// TwinCAT 3 PLC project Steinemann
// Title: CalmarProductSteinemann
// Company: WIFAG-Polytype
// Author: Wifag//Polytype
// ProjectVersion: 3.0.4
// Description: All rights reserved (c) Wifag//Polytype, Fribourg/Switzerland (2021)
// ProgramVersion: 3.1.4023.0
// CompilerDefines: checks_in_libs
// libraries:
//   CalmarCommons, * (WIFAG-Polytype)
//   CalmarCompDevices, * (WIFAG-Polytype)
//   CalmarCompInkSystem, * (WIFAG-Polytype)
//   CalmarCompPrint, * (WIFAG-Polytype)
//   CalmarCompSystem, * (WIFAG-Polytype)
//   CalmarCompTcpIp, * (WIFAG-Polytype)
//   CmpBitmapPool, * (System)
//   Tc2_EtherCAT, * (Beckhoff Automation GmbH)
//   Tc2_Math, * (Beckhoff Automation GmbH)
//   Tc2_Standard, * (Beckhoff Automation GmbH)
//   Tc2_System, * (Beckhoff Automation GmbH)
//   Tc2_TcpIp, * (Beckhoff Automation GmbH)
//   Tc2_Utilities, * (Beckhoff Automation GmbH)
//   Tc3_JsonXml, * (Beckhoff Automation GmbH)
//   VisuDialogs, * (System)
// project tree:
//   DUTs/ADS/ ST_ADS_CLEAN_AXIS.TcDUT, ST_ADS_CLEAN_PROCESS.TcDUT, ST_ADS_DFOIL.TcDUT, ST_ADS_DRYER.TcDUT, ST_ADS_DVTSHEETALIGNMENT.TcDUT, ST_ADS_MOTION_CONTROLLER.TcDUT, ST_ADS_MOTION_SYSTEM.TcDUT, ST_ADS_MOTION_XYR_CONTROLLER.TcDUT, ST_ADS_MOTION_XYR_SYSTEM.TcDUT, ST_ADS_SECURITY.TcDUT
//   DUTs/Camera/ EN_CAMERA_TEACH.TcDUT, E_CameraDevice.TcDUT, E_CameraMode.TcDUT, E_DeformationType.TcDUT, ST_ADS_CAMERA.TcDUT, ST_CameraPoint.TcDUT, ST_CAMERA_CORRECTION_QV.TcDUT, ST_CAMERA_RESULT.TcDUT, ST_CAMERA_TEACH_QV.TcDUT, ST_CORRECTION_POINT.TcDUT, ST_TeachPoint.TcDUT
//   DUTs/CleaningStation/ EN_CLEANING_OP.TcDUT, EN_Cleaning_State.TcDUT, EN_EL7201_STATE.TcDUT, EN_EL7342_STATE.TcDUT, ST_CH_MVT_STATUS.TcDUT, ST_CLEANING_DEV_CMD.TcDUT, ST_CLEANING_DEV_STATUS.TcDUT, ST_CU_STATUS.TcDUT, ST_MANUAL_CMD.TcDUT, ST_PU_STATUS.TcDUT, ST_SPEEDS.TcDUT
//   DUTs/ EN_MSG_LIST.TcDUT, ST_DFOIL_RECORD.TcDUT, ST_SENSOR_COMPARISON.TcDUT
//   / GlobalTextList.TcGTLO, ImagePool_Steinemann.TcIPO (not stored), Visualization Manager.TcVMO (not stored)
//   GVLs/ EC_DefGrid.TcGVL, GVL_Camera.TcGVL, GVL_Deformation.TcGVL, GVL_WEU.TcGVL, GVL_Maxliner.TcGVL
//   POUs/Machine/CleaningStation/ADS/ FB_ADS_CleanAxis.TcPOU, FB_ADS_CleanProcess.TcPOU
//   POUs/Machine/CleaningStation/ FB_CappingCommand.TcPOU, FB_CH_MOTION_CTRL.TcPOU, FB_CH_PROCESS_CTRL.TcPOU, FB_CleanDevice.TcPOU, FB_CleaningMotorAxisCH.TcPOU, FB_CleaningMotorAxisCU.TcPOU, FB_CleaningMotorAxisPU.TcPOU, FB_CleaningProcess.TcPOU, FB_CleaningProcessStateBase.TcPOU, FB_CleaningProcessStateCapping.TcPOU, FB_CleaningProcessStateCappingExit.TcPOU, FB_CleaningProcessStateCleaning.TcPOU, FB_CleaningProcessStateError.TcPOU, FB_CleaningProcessStateInit.TcPOU, FB_CleaningProcessStateProduction.TcPOU, FB_CleaningProcessStateService.TcPOU, FB_CleaningProcessStateWait.TcPOU, FB_CLEANING_PROCESS.TcPOU, FB_Cleaning_ValvePump.TcPOU, FB_CU_MOTION_CTRL.TcPOU, FB_EL7041.TcPOU, FB_EL7201.TcPOU, FB_EL7201_001_AXIS_CTRL.TcPOU, FB_EL7201_AXIS_CTRL.TcPOU, FB_EL7342_AXIS_CTRL.TcPOU, FB_MachineBase.TcPOU, FB_MachineState.TcPOU, FB_MOTOR_SWITCH.TcPOU, FB_PU_MOTION_CTRL.TcPOU, FB_SHUTTER.TcPOU, I_CleanDevice.TcIO, I_CleaningStateCallback.TcIO, I_MachineState.TcIO, I_MachineStateBase.TcIO, _VISU_CleanCH.TcVIS, _VISU_CleanCU.TcVIS, _VISU_CleanProcess.TcVIS, _VISU_CleanPU.TcVIS, _VISU_CleanSequence.TcVIS
//   POUs/Machine/EffectiveEncoderResolutionDetection/ FB_EffectiveEncoderResolutionDetection.TcPOU, _VISU_EffectiveEncoderResolutionDetection.TcVIS
//   POUs/Machine/ExhaustSystem/ FB_ExhaustSystemPrint.TcPOU, _VISU_ExhaustSystemPrint.TcVIS
//   POUs/Machine/ FB_FILTER_MAV_1000.TcPOU, FB_TempLogging_OpcUa.TcPOU
//   POUs/Machine/PowerControl/ FB_PowerControl.TcPOU, _VISU_PowerControl.TcVIS
//   POUs/Machine/SheetDetectSupervision/ FB_SheetDetectSupervision.TcPOU, ST_SheetDetectSupervisionPar.TcDUT (not stored), VISU_SheetDetectSupervision.TcVIS
//   POUs/Machine/UV_LED_Modul/ FB_UvLedModule.TcPOU, _VISU_UvLedModule.TcVIS
//   POUs/Print/Ads/ FB_ADS_CAMERA.TcPOU, FB_ADS_DVTSHEETALIGNMENT.TcPOU
//   POUs/Print/Camera/ FB_CameraBase.TcPOU, FB_CameraDummy.TcPOU, FB_CameraTcpIp.TcPOU, FB_CameraTrigger.TcPOU, FB_MarkCamera.TcPOU, FB_SystronCamera.TcPOU, FB_TcpIpComm.TcPOU, F_DeformationPointAcc_ToString.TcPOU, F_CamPoint_ToString.TcPOU, ImagePool.TcIPO (not stored), I_Camera.TcIO, I_CameraSink.TcIO, I_CameraTrigger.TcIO, I_CameraTriggerDevice.TcIO, _VISU_CameraBase.TcVIS, _VISU_CameraBaseSetting.TcVIS, _VISU_CameraTcpIp.TcVIS, _VISU_CameraTcpIpSetting.TcVIS, _VISU_CameraTrigger.TcVIS, _VISU_DeformationPoint.TcVIS, _VISU_MarkCamera.TcVIS (not stored), _VISU_SystronCamera.TcVIS
//   POUs/Print/Camera/LineCamera/ FB_LineCamera.TcPOU, FB_LineCamera106.TcPOU, FB_LineCamera76.TcPOU, FB_LineCamera585.TcPOU, _VISU_LineCamera.TcVIS
//   POUs/Print/Camera/MarkCameraWEU/ E_MarkMode.TcTLEO, FB_MarkCamera_WEU.TcPOU, FB_MarkDefinition.TcPOU, FB_MarkDetection.TcPOU, I_MarkDefinition.TcIO (not stored), ST_MarkDefinition.TcDUT (not stored), ST_MarkState.TcDUT, ST_MarkView.TcDUT (not stored), ST_RepeatHistory.TcDUT (not stored), TL_MarkMode.TcTLO (not stored), _VISU_MarkCamera_WEU.TcVIS, _VISU_MarkDefinition.TcVIS, _VISU_MarkDefinition_Details.TcVIS (not stored), _VISU_MarkDetection.TcVIS, _VISU_MarkDetection_Trigger.TcVIS (not stored), _VISU_MarkHistory.TcVIS, _VISU_MarkHistoryEntry.TcVIS, _VISU_MarkModes.TcVIS, _VISU_MarkOrientation.TcVIS (not stored), _VISU_MarkOverview.TcVIS, _VISU_MarkTriangle.TcVIS (not stored), _VISU_MarkTriangle_Detail.TcVIS (not stored), _VISU_MarkViewMini.TcVIS, _VISU_RepeatHistory.TcVIS (not stored), _VISU_RepeatHistoryEntry.TcVIS
//   POUs/Print/Camera/Obsolete/ FB_CAMERA_TRIGGER.TcPOU
//   POUs/Print/DefGrid/ E_DeformationStep.TcTLEO, FB_ContainerDefGrid.TcPOU, FB_CTManagerDefGrid.TcPOU, FB_CTTrackerView.TcPOU, FB_DeformationPointFIFO.TcPOU, FB_DropSpeedComp.TcPOU, FB_FineAlignement.TcPOU, FB_ImageDeformation.TcPOU, FB_DefGridParamMediator.TcPOU, FB_PointCorr.TcPOU, FB_PrintOverview.TcPOU, FB_PrintPositionDmax.TcPOU, FB_ProdManager_DMAX.TcPOU, FB_PythonDeformation.TcPOU, FB_PythonInterface.TcPOU, FB_GridDataExporter.TcPOU, FB_StartPositionDummy.TcPOU, FB_WorkerDefGrid.TcPOU, FB_WorkerDefGrid_Camera.TcPOU, FB_WorkerDefGrid_Deformation.TcPOU, FB_WorkerDefGrid_Delete.TcPOU, FB_WorkerDefGrid_Inspection.TcPOU, FB_WorkerDefGrid_Print.TcPOU, FB_WorkerDefGrid_Python.TcPOU, FB_WorkerDefGrid_Verify.TcPOU, F_EncoderSpeedComp.TcPOU, F_MeterToSubPixelReal.TcPOU (not stored), I_DeformationHandler.TcIO, I_GridPointCorrection.TcIO, I_Module.TcIO, I_ParamMediator.TcIO, I_ProdManager.TcIO, ST_CameraGridSettings.TcDUT, ST_CameraPointTbl.TcDUT (not stored), ST_DeformationPointTbl.TcDUT, ST_GridPointUI.TcDUT, ST_WorkerDefGrid_CTData.TcDUT
//   POUs/Print/DefGrid/_Test/ E_GridTypeSelection.TcTLEO, Txt_GridTypeSelection.TcTLO
//   POUs/Print/DefGrid/_VISU_Templates/ E_DeformationType.TcTLO, _VISU_ContainerDefGrid.TcVIS, _VISU_CTsFlow.TcVIS, _VISU_CTTrackerFlow.TcVIS, _VISU_CT_Details.TcVIS, _VISU_DefGridTable.TcVIS, _VISU_DefGridTable_raw.TcVIS, _VISU_FineAlignment.TcVIS, _VISU_GridPointView.TcVIS (not stored), _VISU_ImageDeformation.TcVIS (not stored), _VISU_PlacementXY.TcVIS (not stored), _VISU_PlacementXY_puc.TcVIS (not stored), _VISU_PlacementXY_cross.TcVIS (not stored), _VISU_PmPosition.TcVIS (not stored), _VISU_PrintPositionDmax.TcVIS (not stored), _VISU_DropSpeedComp_Setup.TcVIS, _VISU_ProductionOverview.TcVIS (not stored), _VISU_StartPositionDummy.TcVIS (not stored), _VISU_WorkerDefGrid.TcVIS (not stored), _VISU_WorkerDefGrid_Camera.TcVIS (not stored), _VISU_WorkerDefGrid_Deformation.TcVIS (not stored), _VISU_WorkerDefGrid_Delete.TcVIS (not stored), _VISU_WorkerDefGrid_Print.TcVIS (not stored), _VISU_WorkerDefGrid_Python.TcVIS (not stored), _VISU_WorkerDefGrid_small.TcVIS (not stored), _VISU_WorkerDefGrid_Verify.TcVIS (not stored), _VISU_WorkerDefGrid_VerifyDetail.TcVIS (not stored), _VISU_CTGridExporter.TcVIS, _VISU_WorkerDefGrid_VerifyHistory.TcVIS (not stored)
//   POUs/Print/Global/ I_PrintGlobal.TcIO
//   POUs/Print/Maxliner/ FB_PrintModule_Maxliner.TcPOU, FB_PrintModule_Maxliner_View.TcPOU, _VISU_PmEnable_Maxliner.TcVIS, _VISU_Pm_Maxliner_ImgLengthCheck.TcVIS, _VISU_Pm_Maxliner_Worker.TcVIS, _VISU_Pm_Maxliner_mini_Worker.TcVIS, _VISU_Pm_Maxliner_Debug.TcVIS, _VISU_Pm_Maxliner.TcVIS, _VISU_Pm_Maxliner_Settings.TcVIS
//   POUs/Print/Module/ FB_PrintModule_Base.TcPOU, ST_CassetteSetup.TcDUT, ST_CassetteSetup_Ink.TcDUT, ST_CassetteSetup_Print.TcDUT, ST_MappingDefinition.TcDUT, ST_ModuleMachineInterface_IN.TcDUT, ST_ModuleMachineInterface_OUT.TcDUT
//   POUs/Print/Module/_VISU_Templates/ _VISU_PmEnable.TcVIS (not stored), _VISU_PmEnable_1Worker.TcVIS (not stored), _VISU_Pm_Base_Settings.TcVIS (not stored), _VISU_Pm_MachineIn.TcVIS (not stored), _VISU_Pm_MachineOut.TcVIS (not stored)
//   POUs/Print/obsolete/ FB_DRIFTCONTROL.TcPOU, FB_START_POS_DETECT_WEU.TcPOU, ST_CassetteSetup_PrintAds.TcDUT (excluded from build)
//   POUs/Print/WEU/ FB_PrintModule_WEU.TcPOU, FB_PrintModule_WEU_View.TcPOU, FB_WorkerDefGrid_Print_WEU.TcPOU, _VISU_PmImgLengthCheck.TcVIS, _VISU_Pm_WEU_Debug.TcVIS, _VISU_Pm_WEU_Settings.TcVIS, _VISU_Pm_WEU.TcVIS, _VISU_Pm_WEU_1Worker.TcVIS, _VISU_Pm_WEU_mini.TcVIS, _VISU_Pm_WEU_mini_1Worker.TcVIS, _VISU_Pm_WEU_Worker.TcVIS, _VISU_WorkerPrint_WEU.TcVIS
//   Version/ Global_Version.TcGVL

// ---- DUTs/ADS/ST_ADS_CLEAN_AXIS.TcDUT
TYPE ST_ADS_CLEAN_AXIS :
(*************************************************************************************************)
(*  FILENAME:    ST_ADS_CLEAN_AXIS.EXP                                                           *)
(*  PROJECT:     CALMAR PUPLC                                                                    *)
(*  COPYRIGHT:   All rights reserved (c) Wifag//Polytype, Fribourg/Switzerland (2016)            *)
(*  ENVIRONMENT: TwinCAT PLC                                                                     *)
(*  VERSION:     <version>                                                                       *)
(*************************************************************************************************)
(*  DESCRIPTION:                                                                   <description> *)
(*     User commands from ADS and info feedback to ADS  for cleaning station axis.               *)
(*                                                                                </description> *)
(*************************************************************************************************)

STRUCT
  iO_Version            : INT :=  010001;   (*1.0.1*)
  aO_Type               : STRING := 'Axis';
  aO_Name               : STRING := '';
  sO_Message            : ST_ADS_MSG_IF;

  bI_FaultAck           : BOOL := FALSE;

  (*Manual Move, only possible when in maintenance and manual mode*)
  bI_ManualMove         : BOOL := FALSE;  (*Active as long as true*)
  bO_ManualMoveCanEx    : BOOL := FALSE;
  bO_ManualMovekExec    : BOOL := FALSE;
  fI_ManualTargetPos    : REAL := 0.0;

  (*Current axis position*)
  sO_AxisPosition       : ST_VAR_OUT_REAL;

  wO_ErrorCode          : WORD;
  bO_Busy               : BOOL;
  bO_Ready              : BOOL;
  bO_Error              : BOOL;
END_STRUCT
END_TYPE

// ---- DUTs/ADS/ST_ADS_CLEAN_PROCESS.TcDUT
TYPE ST_ADS_CLEAN_PROCESS :
(*************************************************************************************************)
(*  FILENAME:    ST_ADS_CLEAN_PROCESS                                                            *)
(*  PROJECT:     CALMAR PUPLC                                                                    *)
(*  COPYRIGHT:   All rights reserved (c) Wifag//Polytype, Fribourg/Switzerland (2016)            *)
(*  ENVIRONMENT: TwinCAT PLC                                                                     *)
(*  VERSION:     <version>                                                                       *)
(*************************************************************************************************)
(*  DESCRIPTION:                                                                   <description> *)
(*     User commands from ADS and info feedback to ADS for cleaning station axis.                *)
(*                                                                                </description> *)
(*************************************************************************************************)

STRUCT
  iO_Version                 : INT :=  010001;  (*1.0.1*)
  aO_Type                    : STRING := 'CleanProcess';
  aO_Name                    : STRING :='';
  sO_Message                 : ST_ADS_MSG_IF;
                             
  (*User commands - Trigger operation*)
  bI_StartCapping            : BOOL := FALSE;
  bO_StartCappingCanEx       : BOOL := FALSE;
  bO_StartCappingExec        : BOOL := FALSE;
                             
  bI_StopCapping             : BOOL := FALSE;
  bO_StopCappingCanEx        : BOOL := FALSE;
  bO_StopCappingExec         : BOOL := FALSE;
                             
  bI_Purge                   : BOOL := FALSE;
  bO_PurgeCanEx              : BOOL := FALSE;
  bO_PurgeExec               : BOOL := FALSE;
                             
  bI_Clean                   : BOOL := FALSE;
  bO_CleanCanEx              : BOOL := FALSE;
  bO_CleanExec               : BOOL := FALSE;
                             
  bI_Maintenance             : BOOL := FALSE;
  bO_MaintenanceCanEx        : BOOL := FALSE;
  bO_MaintenanceExec         : BOOL := FALSE;
                             
  bI_OpenShutter             : BOOL := FALSE;
  bO_OpenShutterCanEx        : BOOL := FALSE;
  bO_OpenShutterExec         : BOOL := FALSE;
                             
  bI_Abort                   : BOOL := FALSE;
  bO_AbortCanEx              : BOOL := FALSE;
  bO_AbortExec               : BOOL := FALSE;

  bI_AcknowledgeError        : BOOL := FALSE;
  bO_AcknowledgeErrorCanEx   : BOOL := FALSE;
  bO_AcknowledgeErrorExec    : BOOL := FALSE;

  (*User settings - State operation*)
  bI_AutoMode                : BOOL := TRUE;  (*del*)
  bI_CleanAfterCapp          : BOOL := FALSE;
  bI_CleanAfterPurge         : BOOL := FALSE;
  bI_PurgeAfterCapp          : BOOL := FALSE; (*del*)
  bI_MaintenanceMode         : BOOL := FALSE;
                             
  (*Flags*)                  
  bO_Busy                    : BOOL;
  bO_Ready                   : BOOL;
  bO_ServiceEnabled          : BOOL;
  bO_AxisProcessMovingVisible: BOOL := TRUE;  (*Cleaning process axis moving is shown at PUC*)
                             
  (*Message Queue - TODO update*)
  bI_FaultAck                : BOOL := FALSE;
  wO_ErrorCode               : WORD;
END_STRUCT
END_TYPE

// ---- DUTs/ADS/ST_ADS_DFOIL.TcDUT
TYPE ST_ADS_DFOIL :
(*************************************************************************************************)
(*  FILENAME:    ST_ADS_DFOIL                                                                    *)
(*  PROJECT:     CALMAR PUPLC                                                                    *)
(*  COPYRIGHT:   All rights reserved (c) Wifag//Polytype, Fribourg/Switzerland (2019)            *)
(*  ENVIRONMENT: TwinCAT PLC                                                                     *)
(*  VERSION:     <version>                                                                       *)
(*************************************************************************************************)
(*  DESCRIPTION:                                                                   <description> *)
(*    ADS structure dFoil system.                                                                *)
(*                                                                                </description> *)
(*************************************************************************************************)

STRUCT
  iO_Version         : INT    := 010000;  (*1.0.0*)
  aO_Type            : STRING := 'dFoil';
  aO_Name            : STRING := 'dFoil';

  bI_Enable          : BOOL := TRUE;      (*Enable this device*)
  iO_MaxNbRecords    : UINT  := SIZEOF(sI_dFoilUsagePos) / SIZEOF(sI_dFoilUsagePos[1]);

  iI_UsedNbRecords   : UINT;
  sI_dFoilUsagePos   : ARRAY[1..20] OF ST_DFOIL_RECORD;
END_STRUCT
END_TYPE

// ---- DUTs/ADS/ST_ADS_DRYER.TcDUT
TYPE ST_ADS_DRYER :
(*************************************************************************************************)
(*  FILENAME:    ST_ADS_DRYER.EXP                                                                *)
(*  PROJECT:     CALMAR PUPLC                                                                    *)
(*  COPYRIGHT:   All rights reserved (c) Wifag//Polytype, Fribourg/Switzerland (2016)            *)
(*  ENVIRONMENT: TwinCAT PLC                                                                     *)
(*  VERSION:     <version>                                                                       *)
(*************************************************************************************************)
(*  DESCRIPTION:                                                                   <description> *)
(*     ADS structure for dryer.                                                                  *)
(*                                                                                </description> *)
(*************************************************************************************************)

STRUCT
  iO_Version                  : INT    := 010001;             (*1.0.1*)
  aO_Type                     : STRING := 'Dryer';
  aO_Name                     : STRING := 'DRYER';
  sO_Message                  : ST_ADS_MSG_IF;                (*Messaging*)

  (*I*)
  bI_Enable                   : BOOL := TRUE;                 (*Enable this device*)

  sI_PositionX                : ST_VAR_IN_DINT;               (*Actual position of the dryer on the axis, in micro meters*)
  sI_StartPositionX           : ST_VAR_IN_DINT;               (*Actual position of the dryer on the axis, in micro meters*)

  (*O*)
  cO_StatusDryer              : BYTE;                         (*Bit0:  1h: exist
                                                                Bit1:  2h: enabled
                                                                Bit2:  4h: dryer activ
                                                                Bit3:  8h: warning
                                                                Bit4: 10h: error*)
END_STRUCT
END_TYPE

// ---- DUTs/ADS/ST_ADS_DVTSHEETALIGNMENT.TcDUT
TYPE ST_ADS_DVTSHEETALIGNMENT :
(*************************************************************************************************)
(*  FILENAME:     ST_ADS_DVTSHEETALIGNMENT.EXP                                                   *)
(*  PROJECT:      CALMAR Print System                                                            *)
(*  COPYRIGHT:    Wifag//Polytype Fribourg                                                       *)
(*  ENVIRONMENT:  TwinCAT PLC / CoDeSys                                                          *)
(*  VERSION:      1.0                                                                            *)
(*  DESCRIPTION:  User settings for DVT sheet alignment                                          *)
(*                                                                                               *)
(*  AUTHOR:       FAF                                                                            *)
(*************************************************************************************************)
(*  MODIFICATIONS:                                                                               *)
(*************************************************************************************************)
(*  Date      Author  Comments                                                                   *)
(*  30.04.14  FAF     Created for general use                                                    *)
(*                                                                                               *)
(*************************************************************************************************)

STRUCT
  iO_Version         : INT :=  010010;  (*1.0.10*)
  aO_Type            : STRING := 'DvtSheetAlignment';
  aO_Name            : STRING :='';
  sO_Message         : ST_ADS_MSG_IF;

  (*In*)
  bI_Enable          : BOOL := FALSE;   (*Enable processing*)

  bI_UsePrintMark    : BOOL := TRUE;    (*Enable processing of print marks*)
  sI_PrintMarkSizeX  : ST_VAR_IN_REAL;  (*Print mark X size [mm]*)
  sI_PrintMarkSizeY  : ST_VAR_IN_REAL;  (*Print mark Y size [mm]*)

  sI_HeadGap         : ST_VAR_IN_REAL;  (*Gap between head and substrate [mm]*)

  lI_SegmentSize     : UDINT;           (*Distance between two images in pixel*)
  lI_SegmentCount    : UDINT;           (*Number of images*)
  fI_SegmentAngle    : REAL;            (*Angle between two segments in deg*)

  sI_DeltaX          : ST_VAR_IN_REAL;  (*X offset between camera marks [mm]*)

  bI_IsMaintenanceJob: BOOL;            (*Maintenance job: disable shift and rotation*)

  (*Out*)
  sO_CurrentAngle    : ST_VAR_OUT_REAL; (*Last measured angle in deg*)
  lO_CurrentYShift   : UDINT;           (*Last measured Y Shift in Pixel*)

  bO_RangeErrorAngle : BOOL;            (*Measured angle out of range*)
  bO_RangeErrorShift : BOOL;            (*Measured shift out of range*)
END_STRUCT
END_TYPE

// ---- DUTs/ADS/ST_ADS_MOTION_CONTROLLER.TcDUT
TYPE ST_ADS_MOTION_CONTROLLER :
(*************************************************************************************************)
(*  FILENAME:    ST_ADS_MOTION_CONTROLLER.EXP                                                    *)
(*  PROJECT:     CALMAR PUPLC                                                                    *)
(*  COPYRIGHT:   All rights reserved (c) Wifag//Polytype, Fribourg/Switzerland (2016)            *)
(*  ENVIRONMENT: TwinCAT PLC                                                                     *)
(*  VERSION:     <version>                                                                       *)
(*************************************************************************************************)
(*  DESCRIPTION:                                                                   <description> *)
(*     Add description                                                                           *)
(*                                                                                </description> *)
(*************************************************************************************************)

STRUCT
  iO_Version        : INT :=  010000;  (*1.0.0*)
  aO_Type           : STRING := 'MotionController';
  aO_Name           : STRING := 'MotionController';

END_STRUCT
END_TYPE

// ---- DUTs/ADS/ST_ADS_MOTION_SYSTEM.TcDUT
TYPE ST_ADS_MOTION_SYSTEM :
(*************************************************************************************************)
(*  FILENAME:    ST_ADS_MOTION_SYSTEM.EXP                                                        *)
(*  PROJECT:     CALMAR PUPLC                                                                    *)
(*  COPYRIGHT:   All rights reserved (c) Wifag//Polytype, Fribourg/Switzerland (2016)            *)
(*  ENVIRONMENT: TwinCAT PLC                                                                     *)
(*  VERSION:     <version>                                                                       *)
(*************************************************************************************************)
(*  DESCRIPTION:                                                                   <description> *)
(*     Add description                                                                           *)
(*                                                                                </description> *)
(*************************************************************************************************)

STRUCT
  iO_Version        : INT :=  010000;  (*1.0.0*)
  aO_Type           : STRING := 'MotionSystem';
  aO_Name           : STRING := 'MotionSystem';

END_STRUCT
END_TYPE

// ---- DUTs/ADS/ST_ADS_MOTION_XYR_CONTROLLER.TcDUT
TYPE ST_ADS_MOTION_XYR_CONTROLLER :
(*************************************************************************************************)
(*  FILENAME:    ST_ADS_MOTION_XYR_CONTROLLER.EXP                                                *)
(*  PROJECT:     CALMAR PUPLC                                                                    *)
(*  COPYRIGHT:   All rights reserved (c) Wifag//Polytype, Fribourg/Switzerland (2016)            *)
(*  ENVIRONMENT: TwinCAT PLC                                                                     *)
(*  VERSION:     <version>                                                                       *)
(*************************************************************************************************)
(*  DESCRIPTION:                                                                   <description> *)
(*     Add description                                                                           *)
(*                                                                                </description> *)
(*************************************************************************************************)

STRUCT
  iO_Version        : INT :=  010000;  (*1.0.0*)
  aO_Type           : STRING := 'MotionXyrController';
  aO_Name           : STRING := 'MotionXYRController';

  aO_IpAddress      : STRING;

END_STRUCT
END_TYPE

// ---- DUTs/ADS/ST_ADS_MOTION_XYR_SYSTEM.TcDUT
TYPE ST_ADS_MOTION_XYR_SYSTEM :
(*************************************************************************************************)
(*  FILENAME:    ST_ADS_MOTION_XYR_SYSTEM.EXP                                                    *)
(*  PROJECT:     CALMAR PUPLC                                                                    *)
(*  COPYRIGHT:   All rights reserved (c) Wifag//Polytype, Fribourg/Switzerland (2016)            *)
(*  ENVIRONMENT: TwinCAT PLC                                                                     *)
(*  VERSION:     <version>                                                                       *)
(*************************************************************************************************)
(*  DESCRIPTION:                                                                   <description> *)
(*     Add description                                                                           *)
(*                                                                                </description> *)
(*************************************************************************************************)

STRUCT
  iO_Version        : INT :=  010000;  (*1.0.0*)
  aO_Type           : STRING := 'MotionXyrSystem';
  aO_Name           : STRING := 'MotionXYRSystem';

  iO_Elevation      : DINT;
  iO_Rotation       : DINT;
  sI_PositionX      : ST_VAR_IN_DINT;

END_STRUCT
END_TYPE

// ---- DUTs/ADS/ST_ADS_SECURITY.TcDUT
TYPE ST_ADS_SECURITY :
(*************************************************************************************************)
(*  FILENAME:    ST_ADS_SECURITY.EXP                                                             *)
(*  PROJECT:     CALMAR PUPLC                                                                    *)
(*  COPYRIGHT:   All rights reserved (c) Wifag//Polytype, Fribourg/Switzerland (2016)            *)
(*  ENVIRONMENT: TwinCAT PLC                                                                     *)
(*  VERSION:     <version>                                                                       *)
(*************************************************************************************************)
(*  DESCRIPTION:                                                                   <description> *)
(*     ADS structure for security.                                                               *)
(*                                                                                </description> *)
(*************************************************************************************************)

STRUCT
  iO_Version                  : INT    := 010000;             (*1.0.0*)
  aO_Type                     : STRING := 'Security';
  aO_Name                     : STRING := 'SECURITY';
  sO_Message                  : ST_ADS_MSG_IF;                (*Messaging*)

  (*I*)
  bI_Enable                   : BOOL := TRUE;                 (*Enable this device*)

  (*O*)
  bO_ErrorEmergencyStopButton : BOOL;                         (*Emergency stop*)
  bO_ErrorDoorMonitoring      : BOOL;                         (*Doors*)
  bO_ErrorCheckSumFuses       : BOOL;                         (*Fuses*)
  bO_ErrorExternalSecurity    : BOOL;                         (*Security from external*)
END_STRUCT
END_TYPE

// ---- DUTs/Camera/EN_CAMERA_TEACH.TcDUT
TYPE EN_CAMERA_TEACH :
(*************************************************************************************************)
(*  FILENAME:    EN_CAMERA_TEACH                                                                 *)
(*  PROJECT:     CALMAR PUPLC                                                                    *)
(*  COPYRIGHT:   All rights reserved (c) Wifag//Polytype, Fribourg/Switzerland (2018)            *)
(*  ENVIRONMENT: TwinCAT PLC                                                                     *)
(*  VERSION:     <version>                                                                       *)
(*************************************************************************************************)
(*  DESCRIPTION:                                                                   <description> *)
(*    Enumeration for camera teach.                                                              *)
(*                                                                                </description> *)
(*************************************************************************************************)

(
  eTeachInit         := 0,
  eTeachStart        := 1,
  eTeachCompleted    := 2,
  eTeachCanceled     := 3,
  eTeachError        := 4
);
END_TYPE

// ---- DUTs/Camera/E_CameraDevice.TcDUT
{attribute 'qualified_only'}
{attribute 'strict'}
{attribute 'to_string'}
TYPE E_CameraDevice :
(
  SheetDetect              := 0,   // SheetDetect
  PrintMark                := 1,   // PrintMark
  Scanner                  := 2,   // Scanner
  ScannerWithoutBackground := 3    // ScannerWithoutBackground
);
END_TYPE

// ---- DUTs/Camera/E_CameraMode.TcDUT
{attribute 'qualified_only'}
{attribute 'strict'}
{attribute 'to_string'}
TYPE E_CameraMode :
(
  NoCorrection := 0,   // NoCorrection
  XYR          := 1,   // XYR
  Live         := 2,   // Live deformation
  Trend        := 3,   // Live deformation with trend
  Auto         := 4    // Auto
);
END_TYPE

// ---- DUTs/Camera/E_DeformationType.TcDUT
{attribute 'qualified_only'}
{attribute 'to_string'}
TYPE E_DeformationType :
(
  NoDeformation   := 0,   // NoCorrection
  ScriptGrid      := 1,   // Py script (live)
  ScriptGridTrend := 2,   // Py script (live with trend)
  LocalMarks1D    := 3    // Plc generated with 1D marks
)  UINT;
END_TYPE

// ---- DUTs/Camera/ST_ADS_CAMERA.TcDUT
TYPE ST_ADS_CAMERA :
(*************************************************************************************************)
(*  FILENAME:    ST_ADS_CAMERA                                                                   *)
(*  PROJECT:     CALMAR PUPLC                                                                    *)
(*  COPYRIGHT:   All rights reserved (c) Wifag//Polytype, Fribourg/Switzerland (2018)            *)
(*  ENVIRONMENT: TwinCAT PLC                                                                     *)
(*  VERSION:     <version>                                                                       *)
(*************************************************************************************************)
(*  DESCRIPTION:                                                                   <description> *)
(*    ADS structure for camera (Systron, QualiVision).                                           *)
(*                                                                                </description> *)
(*************************************************************************************************)

STRUCT
  iO_Version                : UINT    := 010300;  (*1.3.0*)
  aO_Type                   : STRING := 'Camera';
  aO_Name                   : STRING := 'Camera';
  sO_Message                : ST_ADS_MSG_IF;

  (*In*)
  bI_Enable                 : BOOL := TRUE;      (*Enable this device*)

  eI_CameraDevice           : E_CameraDevice;    (*Camera device*)
  eI_CameraMode             : E_CameraMode;      (*Camera mode*)

  eI_TeachProgress          : EN_CAMERA_TEACH;   (*Teach progress*)
  sI_TeachPointsQV          : ARRAY[1..GVL_Camera.cC_QUALIVISION_MAX_NB_MARKS] OF ST_CAMERA_TEACH_QV;
  
  sI_CorrectionPointIndication: ARRAY[1..4] OF ST_CORRECTION_POINT;

  (*Out*)
  iO_MaxNbMarksQV           : INT := GVL_Camera.cC_QUALIVISION_MAX_NB_MARKS; 
  sO_PointsReadQV           : ST_COMMAND_PLC;    (*New points read by QualiVision*)
  iO_AvailableNbReadPointQV : INT; 
  sO_ReadPointsQV           : ARRAY[1..GVL_Camera.cC_QUALIVISION_MAX_NB_MARKS] OF ST_CAMERA_CORRECTION_QV;

END_STRUCT
END_TYPE

// ---- DUTs/Camera/ST_CameraPoint.TcDUT
TYPE ST_CameraPoint :
STRUCT
  (*Valus from camera [px/4800dpi]*)
  id                  : UDINT := 0;     (*mark id*)
  x_ref               : DINT := 0;      (*Referenz x deviation [px/4800dpi]*)
  y_ref               : DINT := 0;      (*Referenz y deviation [px/4800dpi]*)
  lx                  : DINT := 0;      (*Referenz in picture x deviation [px/4800dpi]*)
  ly                  : DINT := 0;      (*Referenz in picture y deviation [px/4800dpi]*)
  valid               : BOOL := FALSE;  (*TRUE = PASS, FALSE = FAIL*)
  x                   : DINT := 0;      (*x deviation [px/4800dpi]*)
  y                   : DINT := 0;      (*y deviation [px/4800dpi]*)
END_STRUCT
END_TYPE

// ---- DUTs/Camera/ST_CAMERA_CORRECTION_QV.TcDUT
TYPE ST_CAMERA_CORRECTION_QV :
(*************************************************************************************************)
(*  FILENAME:    ST_CAMERA_CORRECTION_QV                                                         *)
(*  PROJECT:     CALMAR PUPLC                                                                    *)
(*  COPYRIGHT:   All rights reserved (c) Wifag//Polytype, Fribourg/Switzerland (2016)            *)
(*  ENVIRONMENT: TwinCAT PLC                                                                     *)
(*  VERSION:     <version>                                                                       *)
(*************************************************************************************************)
(*  DESCRIPTION:                                                                   <description> *)
(*    Correction of smart camera QualiVision for PUC.                                            *)
(*                                                                                </description> *)
(*************************************************************************************************)

STRUCT
  (*PUC correction points [mm]*)
  valid               : BOOL := FALSE;  (*TRUE = PASS, FALSE = FAIL*)
  PaddingByte01       : BYTE;           (*PUC needs it for stream reading. TC3 uses 8 byte alignment.*)
  PaddingByte02       : BYTE;           (*PUC needs it for stream reading. TC3 uses 8 byte alignment.*)
  PaddingByte03       : BYTE;           (*PUC needs it for stream reading. TC3 uses 8 byte alignment.*)
  x_origin            : REAL := 0;      (*Referenz x origin [mm]*)
  y_origin            : REAL := 0;      (*Referenz y origin [mm]*)
  x_correction        : REAL := 0;      (*x correction [mm]*)
  y_correction        : REAL := 0;      (*y correction [mm]*)
  PaddingBytes04      : REAL;           (*PUC needs it for stream reading. TC3 uses 8 byte alignment.*)
END_STRUCT
END_TYPE

// ---- DUTs/Camera/ST_CAMERA_RESULT.TcDUT
TYPE ST_CAMERA_RESULT :
(*************************************************************************************************)
(*  FILENAME:    ST_CAMERA_RESULT.EXP                                                            *)
(*  PROJECT:     CALMAR PUPLC                                                                    *)
(*  COPYRIGHT:   All rights reserved (c) Wifag//Polytype, Fribourg/Switzerland (2016)            *)
(*  ENVIRONMENT: TwinCAT PLC                                                                     *)
(*  VERSION:     <version>                                                                       *)
(*************************************************************************************************)
(*  DESCRIPTION:                                                                   <description> *)
(*    Output of smart camera Systron.                                                            *)
(*                                                                                </description> *)
(*************************************************************************************************)

STRUCT
  x_ref               : REAL := 0;      (*Referenz x deviation [mm]*)
  y_ref               : REAL := 0;      (*Referenz y deviation [mm]*)
  valid               : BOOL := TRUE;   (*TRUE = PASS, FALSE = FAIL*)
  x                   : REAL := 0;      (*x deviation [mm]*)
  y                   : REAL := 0;      (*y deviation [mm]*)
END_STRUCT
END_TYPE

// ---- DUTs/Camera/ST_CAMERA_TEACH_QV.TcDUT
TYPE ST_CAMERA_TEACH_QV :
(*************************************************************************************************)
(*  FILENAME:    ST_CAMERA_TEACH_QV                                                              *)
(*  PROJECT:     CALMAR PUPLC                                                                    *)
(*  COPYRIGHT:   All rights reserved (c) Wifag//Polytype, Fribourg/Switzerland (2016)            *)
(*  ENVIRONMENT: TwinCAT PLC                                                                     *)
(*  VERSION:     <version>                                                                       *)
(*************************************************************************************************)
(*  DESCRIPTION:                                                                   <description> *)
(*    Teach points for smart camera QualiVision from PUC.                                        *)
(*                                                                                </description> *)
(*************************************************************************************************)

STRUCT
  x_ref_Print         : REAL := 0;      (*Referenz x deviation [mm]*)
  y_ref_Print         : REAL := 0;      (*Referenz y deviation [mm]*)
END_STRUCT
END_TYPE

// ---- DUTs/Camera/ST_CORRECTION_POINT.TcDUT
TYPE ST_CORRECTION_POINT :
(*************************************************************************************************)
(*  FILENAME:    ST_CORRECTION_POINT                                                             *)
(*  PROJECT:     CALMAR PUPLC                                                                    *)
(*  COPYRIGHT:   All rights reserved (c) Wifag//Polytype, Fribourg/Switzerland (2021)            *)
(*  ENVIRONMENT: TwinCAT PLC                                                                     *)
(*  VERSION:     <version>                                                                       *)
(*************************************************************************************************)
(*  DESCRIPTION:                                                                   <description> *)
(*    PUC correction point indication provided from job, written at print start.                 *)
(*                                                                                </description> *)
(*************************************************************************************************)

STRUCT
  x        : REAL := 0;      (*Correction indication x [mm]*)
  y        : REAL := 0;      (*Correction indication y [mm]*)
  posx     : REAL := 0;      (*Correction location in x [mm]*)
  posy     : REAL := 0;      (*Correction location in y [mm]*)
END_STRUCT
END_TYPE

// ---- DUTs/Camera/ST_TeachPoint.TcDUT
TYPE ST_TeachPoint :
STRUCT
  (*Valus for printer [mm]*)
  id                  : UDINT;           (*point id*)
  x_ref_Print         : LREAL := 0;      (*Referenz x deviation [mm]*)
  y_ref_Print         : LREAL := 0;      (*Referenz y deviation [mm]*)
  x_teach_Print       : LREAL := 0;      (*Teach x deviation [mm]*)
  y_teach_Print       : LREAL := 0;      (*Teach y deviation [mm]*)
  x_Print             : LREAL := 0;      (*x deviation [mm]*)
  y_Print             : LREAL := 0;      (*y deviation [mm]*)
  valid               : BOOL  := FALSE;  (**)
END_STRUCT
END_TYPE

// ---- DUTs/CleaningStation/EN_CLEANING_OP.TcDUT
TYPE EN_CLEANING_OP :
(*************************************************************************************************)
(*  FILENAME:    EN_CLEANING_OP.EXP                                                              *)
(*  PROJECT:     CALMAR PUPLC                                                                    *)
(*  COPYRIGHT:   All rights reserved (c) Polytype AG, Fribourg/Switzerland (2020)                *)
(*  ENVIRONMENT: TwinCAT PLC                                                                     *)
(*  VERSION:     <version>                                                                       *)
(*************************************************************************************************)
(*  DESCRIPTION:                                                                   <description> *)
(*     Add description                                                                           *)
(*                                                                                </description> *)
(*************************************************************************************************)
(
  eNOP             := 0,          (*No operation active*)
  eOPCLEAN         := 1,          (*Cleaning*)
  eOPPURGE         := 2,          (*Purging*)
  eOPCAPENTER      := 3,          (*Enter Capping*)
  eOPCAPEXIT       := 4,          (*Exit Capping*)
  eOPMAINT         := 5,          (*Maintenance*)
  eOPSHUTTEROPEN   := 6,          (*Open Shutter*)
  eOPPREPSERVICE   := 7,          (*Prepare cleaning station for servce*)
  eOPENDSERVICE    := 8,          (*End service mode for cleaning station*)
  eOPSTARTUP       := 9,          (*Prepare system for operation*)
  eOPGOTOPROD	     := 10,         (*Prepare system for production*)
  eOPGOTOWAIT	     := 11,					(*Prepare system to production pause*)
  eOPEXITERROR	   := 20					(*Return from Error*)
);
END_TYPE

// ---- DUTs/CleaningStation/EN_Cleaning_State.TcDUT
{attribute 'qualified_only'}
{attribute 'strict'}
TYPE EN_Cleaning_State :
(
	Init        := 0,
	Production  := 1,
	Wait        := 2,
	Service     := 3,
	Capping     := 4,
	CappingExit := 5,
	Cleaning    := 6,
	Error       := 7
);
END_TYPE

// ---- DUTs/CleaningStation/EN_EL7201_STATE.TcDUT
TYPE EN_EL7201_STATE :
(*************************************************************************************************)
(*  FILENAME:    EN_EL7201_STATE.EXP                                                             *)
(*  PROJECT:     CALMAR PUPLC                                                                    *)
(*  COPYRIGHT:   All rights reserved (c) Wifag//Polytype, Fribourg/Switzerland (2016)            *)
(*  ENVIRONMENT: TwinCAT PLC                                                                     *)
(*  VERSION:     <version>                                                                       *)
(*************************************************************************************************)
(*  DESCRIPTION:                                                                   <description> *)
(*     Add description                                                                           *)
(*                                                                                </description> *)
(*************************************************************************************************)
(
  eNotReadyToSwitchON  := 16#0000,
  eSwitchONDisabled    := 16#0040,
  eReadyToSwitchON     := 16#0021,
  eSwitchedON          := 16#0023,
  eEnabled             := 16#0027,
  eFaultReactionActive := 16#000F,
  eFault               := 16#0008,
  eEstopped            := 16#9999
);
END_TYPE

// ---- DUTs/CleaningStation/EN_EL7342_STATE.TcDUT
TYPE EN_EL7342_STATE :
(*************************************************************************************************)
(*  FILENAME:    EN_EL7342_STATE.EXP                                                             *)
(*  PROJECT:     CALMAR PUPLC                                                                    *)
(*  COPYRIGHT:   All rights reserved (c) Wifag//Polytype, Fribourg/Switzerland (2016)            *)
(*  ENVIRONMENT: TwinCAT PLC                                                                     *)
(*  VERSION:     <version>                                                                       *)
(*************************************************************************************************)
(*  DESCRIPTION:                                                                   <description> *)
(*     Add description                                                                           *)
(*                                                                                </description> *)
(*************************************************************************************************)
(
  eReadyToEnable    := 1,
  eReady            := 2,
  eStarted          := 3,
  eFaulty           := 0,
  eEmergencyStopped := 9
);
END_TYPE

// ---- DUTs/CleaningStation/ST_CH_MVT_STATUS.TcDUT
TYPE ST_CH_MVT_STATUS :
(*************************************************************************************************)
(*  FILENAME:    ST_CH_MVT_STATUS                                                                *)
(*  PROJECT:     CALMAR PUPLC                                                                    *)
(*  COPYRIGHT:   All rights reserved (c) Wifag//Polytype, Fribourg/Switzerland (2016)            *)
(*  ENVIRONMENT: TwinCAT PLC                                                                     *)
(*  VERSION:     <version>                                                                       *)
(*************************************************************************************************)
(*  DESCRIPTION:                                                                   <description> *)
(*    Information feedback about the mouvement cycle and the position.                           *)
(*                                                                                </description> *)
(*************************************************************************************************)

STRUCT
  bO_Active                  : BOOL;  (*Cleaning Head is powered up*)
  bO_Ready                   : BOOL;  (*Cleaning Head is ready for new command*)
  bO_Busy                    : BOOL;  (*Cleaning Head has a work in progress*)
  bO_Finished                : BOOL;  (*Cleaning Head is finished*)

  iO_OperationType           : INT;   (*0-Standby ; 1-Cleaning*)

  fO_ClnHead_Position        : REAL;  (*Estimation in mm (speed*time)*)
  bO_Error                   : BOOL;
  wO_FaultCode               : WORD;
END_STRUCT
END_TYPE

// ---- DUTs/CleaningStation/ST_CLEANING_DEV_CMD.TcDUT
TYPE ST_CLEANING_DEV_CMD :
(*************************************************************************************************)
(*  FILENAME:    ST_CLEANING_DEV_CMD.EXP                                                         *)
(*  PROJECT:     CALMAR PUPLC                                                                    *)
(*  COPYRIGHT:   All rights reserved (c) Wifag//Polytype, Fribourg/Switzerland (2016)            *)
(*  ENVIRONMENT: TwinCAT PLC                                                                     *)
(*  VERSION:     <version>                                                                       *)
(*************************************************************************************************)
(*  DESCRIPTION:                                                                   <description> *)
(*     Command for cleaning axis.                                                                *)
(*                                                                                </description> *)
(*************************************************************************************************)

STRUCT
(*Commands*)
  bInit             : BOOL;  (*Initialize operation*)
  bPrep             : BOOL;  (*Prepare operation*)
  bStart            : BOOL;  (*Start operation*)
  bStop             : BOOL;  (*Stop operation*)
  bAbort            : BOOL;  (*Abort operation*)
  bAckError         : BOOL;  (*Acknowledge Error*)

  bAuto             : BOOL;  (*Automatic mode selected*)
  bService          : BOOL;  (*Service mode enabled*)

  eOperation        : EN_CLEANING_OP;  (*Active Operation*)
END_STRUCT
END_TYPE

// ---- DUTs/CleaningStation/ST_CLEANING_DEV_STATUS.TcDUT
TYPE ST_CLEANING_DEV_STATUS :
(*************************************************************************************************)
(*  FILENAME:    ST_CLEANING_DEV_STATUS.EXP                                                      *)
(*  PROJECT:     CALMAR PUPLC                                                                    *)
(*  COPYRIGHT:   All rights reserved (c) Wifag//Polytype, Fribourg/Switzerland (2016)            *)
(*  ENVIRONMENT: TwinCAT PLC                                                                     *)
(*  VERSION:     <version>                                                                       *)
(*************************************************************************************************)
(*  DESCRIPTION:                                                                   <description> *)
(*     Feedback from cleaning axis.                                                              *)
(*                                                                                </description> *)
(*************************************************************************************************)

STRUCT
  bBusy      : BOOL;  (*The axis has a pending command*)
  bReady     : BOOL;  (*The axis is ready for a new command*)
  bError     : BOOL;  (*The axis has an error*)
  bRefKnown  : BOOL;  (*The axis is initialized*)
END_STRUCT
END_TYPE

// ---- DUTs/CleaningStation/ST_CU_STATUS.TcDUT
TYPE ST_CU_STATUS :
(*************************************************************************************************)
(*  FILENAME:    ST_CU_STATUS                                                                    *)
(*  PROJECT:     CALMAR PUPLC                                                                    *)
(*  COPYRIGHT:   All rights reserved (c) Wifag//Polytype, Fribourg/Switzerland (2016)            *)
(*  ENVIRONMENT: TwinCAT PLC                                                                     *)
(*  VERSION:     <version>                                                                       *)
(*************************************************************************************************)
(*  DESCRIPTION:                                                                   <description> *)
(*    Information feedback about the mouvement cycle and the position.                           *)
(*                                                                                </description> *)
(*************************************************************************************************)

STRUCT
  bO_Active                  : BOOL;  (*Cleaning Unit is powered up*)
  bO_Ready                   : BOOL;  (*Cleaning Unit is ready for new command*)
  bO_Busy                    : BOOL;  (*Cleaning Unit has a work in progress*)
  bO_ReferenceKnown          : BOOL;  (*Copy of sensor feedback*)
  fO_Position                : REAL;  (*Processed copy of resolver feedback*)
  bO_InPosition_Cleaning     : BOOL;
  bO_InPosition_Capping      : BOOL;
  bO_InPosition_Purging      : BOOL;
  bO_InPosition_Parking      : BOOL;
  wO_FaultCode               : WORD;
  bO_Error                   : BOOL;
END_STRUCT
END_TYPE

// ---- DUTs/CleaningStation/ST_MANUAL_CMD.TcDUT
TYPE ST_MANUAL_CMD :
(*************************************************************************************************)
(*  FILENAME:    ST_MANUAL_CMD.EXP                                                               *)
(*  PROJECT:     CALMAR PUPLC                                                                    *)
(*  COPYRIGHT:   All rights reserved (c) Wifag//Polytype, Fribourg/Switzerland (2016)            *)
(*  ENVIRONMENT: TwinCAT PLC                                                                     *)
(*  VERSION:     <version>                                                                       *)
(*************************************************************************************************)
(*  DESCRIPTION:                                                                   <description> *)
(*     Structure to regroup the manual command actions and parameter.                            *)
(*                                                                                </description> *)
(*************************************************************************************************)

STRUCT
  fI_Start_position  : REAL;  (*  Position ID for the Upper limit    *)
  fI_Stop_position   : REAL;  (*  Position ID for the lower limit    *)
  bI_Do              : BOOL;  (*  Do action    *)
  bI_Undo            : BOOL;  (*  Undo action    *)
END_STRUCT
END_TYPE

// ---- DUTs/CleaningStation/ST_PU_STATUS.TcDUT
TYPE ST_PU_STATUS :
(*************************************************************************************************)
(*  FILENAME:    ST_PU_STATUS                                                                    *)
(*  PROJECT:     CALMAR PUPLC                                                                    *)
(*  COPYRIGHT:   All rights reserved (c) Wifag//Polytype, Fribourg/Switzerland (2016)            *)
(*  ENVIRONMENT: TwinCAT PLC                                                                     *)
(*  VERSION:     <version>                                                                       *)
(*************************************************************************************************)
(*  DESCRIPTION:                                                                   <description> *)
(*    Information feedback about the mouvement cycle and the position.                           *)
(*                                                                                </description> *)
(*************************************************************************************************)

STRUCT
  bO_Active                  : BOOL;  (*Print Head is powered up*)
  bO_Ready                   : BOOL;  (*Print head is ready for work*)
  bO_Busy                    : BOOL;  (*Print head is busy*)
  fO_Position                : REAL;  (*Processed copy of absolute encoder feedback*)
  bO_InPosition_C1           : BOOL;
  bO_InPosition_C2           : BOOL;
  bO_InPosition_Waiting      : BOOL;
  bO_InPosition_Printing     : BOOL;
  bO_InPosition_Service      : BOOL;
  wO_FaultCode               : WORD;
  bO_Error                   : BOOL;
END_STRUCT
END_TYPE

// ---- DUTs/CleaningStation/ST_SPEEDS.TcDUT
TYPE ST_SPEEDS :
(*************************************************************************************************)
(*  FILENAME:    ST_SPEEDS.EXP                                                                   *)
(*  PROJECT:     CALMAR PUPLC                                                                    *)
(*  COPYRIGHT:   All rights reserved (c) Wifag//Polytype, Fribourg/Switzerland (2016)            *)
(*  ENVIRONMENT: TwinCAT PLC                                                                     *)
(*  VERSION:     <version>                                                                       *)
(*************************************************************************************************)
(*  DESCRIPTION:                                                                   <description> *)
(*     Structure to regroup the speeds parameters of the axis.                                   *)
(*                                                                                </description> *)
(*************************************************************************************************)

STRUCT
  fP_PlaceSpeed    : REAL;  (*  speed for placement mouvement    *)
  fP_WorkSpeed     : REAL;  (*  speed for work mouvement    *)
  fP_ServiceSpeed  : REAL;  (*  speed for maintenance operations    *)
END_STRUCT
END_TYPE

// ---- DUTs/EN_MSG_LIST.TcDUT
TYPE EN_MSG_LIST :
(*************************************************************************************************)
(*  FILENAME:    EN_MSG_LIST.EXP                                                                 *)
(*  PROJECT:     CALMAR PUPLC                                                                    *)
(*  COPYRIGHT:   All rights reserved (c) Wifag//Polytype, Fribourg/Switzerland (2016)            *)
(*  ENVIRONMENT: TwinCAT PLC                                                                     *)
(*  VERSION:     <version>                                                                       *)
(*************************************************************************************************)
(*  DESCRIPTION:                                                                   <description> *)
(*     This block containts the global list for all messages used by `FB_MESSAGE`.               *)
(*                                                                                </description> *)
(*************************************************************************************************)
(
  // start at                       eCStag_MSG_BASE := 10000,
  eC_STAG_CAM_NOTAVAIL                              :=10000,  (*CameraNotAvailable*)
  eC_STAG_CAM_MODE_NOTSUPPORTED                     :=10001,  (*CameraModeNotSupported*)
  eC_STAG_CAM_NOTENGOUGH_TEACH_POINTS               :=10002,  (*CameraNotEnoughTeachPoints*)
  eC_STAG_DEF_SCRIPT_NOT_RUNNING                    :=10003,  (*DeformationScriptNotRunning*)
  eC_STAG_CAM_TEACH_ERROR                           :=10004,  (*CameraTeachError*)
  eC_STAG_IMAGELENGTH_NOT_SUPPORTED                 :=10005,  (*ImageLengthNotSupported*)
  eC_STAG_DEFORMATION_LIMITED                       :=10006   (*DeformationWasLimited (Warning)*)
);
END_TYPE

// ---- DUTs/ST_DFOIL_RECORD.TcDUT
TYPE ST_DFOIL_RECORD :
(*************************************************************************************************)
(*  FILENAME:    ST_DFOIL_RECORD                                                                 *)
(*  PROJECT:     CALMAR PUPLC                                                                    *)
(*  COPYRIGHT:   All rights reserved (c) Wifag//Polytype, Fribourg/Switzerland (2019)            *)
(*  ENVIRONMENT: TwinCAT PLC                                                                     *)
(*  VERSION:     <version>                                                                       *)
(*************************************************************************************************)
(*  DESCRIPTION:                                                                   <description> *)
(*    Record for dFoil system.                                                                   *)
(*                                                                                </description> *)
(*************************************************************************************************)

STRUCT
  lI_StartOffset           : UDINT;       (*Start offset [µm], dFoil not used*)
  lI_PrintedZoneLength     : UDINT;       (*Printed zone length [µm], dFoil used*)
END_STRUCT
END_TYPE

// ---- DUTs/ST_SENSOR_COMPARISON.TcDUT
TYPE ST_SENSOR_COMPARISON :
(*************************************************************************************************)
(*  FILENAME:    ST_SENSOR_COMPARISON.EXP                                                        *)
(*  PROJECT:     CALMAR PUPLC                                                                    *)
(*  COPYRIGHT:   All rights reserved (c) Wifag//Polytype, Fribourg/Switzerland (2016)            *)
(*  ENVIRONMENT: TwinCAT PLC                                                                     *)
(*  VERSION:     <version>                                                                       *)
(*************************************************************************************************)
(*  DESCRIPTION:                                                                   <description> *)
(*    Structure for comparison of mark and camera values.                                        *)
(*                                                                                </description> *)
(*************************************************************************************************)

STRUCT
 	xMark                : DINT;  (*Start position in pixels in Xprint-axis*)
  yMark                : INT;   (*Shift in pixels in Yprint-axis*)
  phiMark              : DINT;  (*Rotation angle*)
 	xCam                 : DINT;  (*Start position in pixels in Xprint-axis*)
  yCam                 : INT;   (*Shift in pixels in Yprint-axis*)
  phiCam               : DINT;  (*Rotation angle*)
 	dx                   : DINT;  (*Start position in pixels in Xprint-axis*)
  dy                   : INT;   (*Shift in pixels in Yprint-axis*)
  dphi                 : DINT;  (*Rotation angle*)
END_STRUCT
END_TYPE

// ---- POUs/Print/Camera/MarkCameraWEU/E_MarkMode.TcTLEO
{attribute 'qualified_only'}
{attribute 'strict'}
{attribute 'to_string'}
TYPE E_MarkMode :
(
	AutoDefault := 0,       // a start mark and all intermediate marks, given by formula
	None        := 1,        // no marks defined, simulate marks
	OneDefault  := 2,       // only one "default* mark at beginning of sheet
  OneTriangle := 3       // only one "old" mark with a rectancular triangle
) UINT := AutoDefault ;
END_TYPE

// ---- POUs/Print/Camera/MarkCameraWEU/ST_MarkState.TcDUT
TYPE ST_MarkState :
STRUCT
  bSet        : BOOL;     // mark was set (detected)
  bMissed     : BOOL;     // mark was missing (+internally generated)
  bInArea     : BOOL;     // mark withing ok area
  dx          : LREAL;    // x displacement [m]
  dy          : LREAL;    // y displacement [m]
  fLengthReal : LREAL;    // real detected mark length [m]
  nPosXReal   : DINT;     // detected position X absolute [SubPx]
  END_STRUCT
END_TYPE

// ---- POUs/Print/DefGrid/E_DeformationStep.TcTLEO
{attribute 'qualified_only'}
{attribute 'strict'}
{attribute 'to_string'}
TYPE E_DeformationStep :
(
  nothing := 0,
  createdScriptContainer := 1,
  cameraStarted := 2,
  cameraDone := 3,
  gridStarted := 4
);
END_TYPE

// ---- POUs/Print/DefGrid/ST_CameraGridSettings.TcDUT
TYPE ST_CameraGridSettings :
STRUCT
  bValid            : BOOL;   // ?
  eCameraMode       : E_CameraMode;
  eDeformationType  : E_DeformationType;  // selected deformation type based on selecte camera and settings
  fGridFeaturePitch : LREAL;  // feature grid picth (cam frame width) [px]
  fDetectToCam      : LREAL;  // distance between detection and camera [m]
END_STRUCT
END_TYPE

// ---- POUs/Print/DefGrid/ST_DeformationPointTbl.TcDUT
(*
  Table representation of a point
*)
TYPE ST_DeformationPointTbl :
STRUCT
  bSet          : BOOL;
  tTime         : T_DCTIME64;
  sPoint        : ST_DeformationPointAccurate;
END_STRUCT
END_TYPE

// ---- POUs/Print/DefGrid/ST_GridPointUI.TcDUT
TYPE ST_GridPointUI :
STRUCT
  valid         : BOOL := 0;      (*valid point?*)
  col           : DINT := 0;      (*point definition*)
  row           : DINT := 0;      (*point definition*)
  x_ref         : LREAL := 0;     (*Referenz x [px]*)
  y_ref         : LREAL := 0;     (*Referenz y [px]*)
  dx            : LREAL := 0;     (*x deviation [px]*)
  dy            : LREAL := 0;     (*y deviation [px]*)
END_STRUCT
END_TYPE

// ---- POUs/Print/DefGrid/ST_WorkerDefGrid_CTData.TcDUT
// workers additional data for all attached CTs
TYPE ST_WorkerDefGrid_CTData :
STRUCT
  fPosRelToAttach : LREAL;    // ct relative position to attach
  nChargedCols : UDINT;       // number of streamed columns of this ct
  nXS : DINT;                 // XS print start position
END_STRUCT
END_TYPE

// ---- POUs/Print/DefGrid/_Test/E_GridTypeSelection.TcTLEO
{attribute 'qualified_only'}
{attribute 'strict'}
{attribute 'to_string'}
TYPE E_GridTypeSelection :
(
  Default             := 0,  // Default deformation based on cam points
  None                := 1,  // No deformation calculated all dx/dy=0
  Test_AllDxFactor    := 2,  // Dx constant for all = factor
  Test_AllDyFactor    := 3,  // Dy constant for all = factor
  Test_DyColFactor    := 4,  // Dy = col * factor (changes by column)
  Test_DxColFactor    := 5,  // Dx = col * factor (changes by column)
  Test_Dx_Row1OnlyFactor := 6   // dx factor only on row1 (test BOF)
) UINT := Default ;
END_TYPE

// ---- POUs/Print/Module/ST_CassetteSetup.TcDUT
TYPE ST_CassetteSetup :
STRUCT
  aName         : T_MaxString;      // module name
  aNameShort    : T_MaxString;      // module name short string
  nIdx          : UDINT;            // module index in Array [1..x]
  nMaschineIdx  : UDINT;            // Module number in machine (station number in machine notation [eg. 3, 4, ...])

  pSetupPrint   : POINTER TO ST_CassetteSetup_Print;  // ref to print settings
  pSetupInk     : POINTER TO ST_CassetteSetup_Ink;    // ref to ink settings
END_STRUCT
END_TYPE

// ---- POUs/Print/Module/ST_CassetteSetup_Ink.TcDUT
TYPE ST_CassetteSetup_Ink :
STRUCT
  // ink settings
  pInkDefinition        : POINTER TO ST_INKDEFINITON;
  pInkHeaderTankGroup   : POINTER TO FB_ADS_HeadertankGroup;
END_STRUCT
END_TYPE

// ---- POUs/Print/Module/ST_CassetteSetup_Print.TcDUT
TYPE ST_CassetteSetup_Print :
STRUCT
  // print settings
  aAmsNetId_Localhost : T_AmsNetID;           // AMS NetID for file access
  aAmsNetId_Io        : T_AmsNetID;           // AMS NetID of EtherCAT master
  nEcatAddr_Pc_Base   : UINT;                 // Base address ethercat slave address of PCs in this module
  pOd                 : POINTER TO FB_OD;     // Pointer to object dictionary of PC
  aCfgPath            : T_MaxString;          // Configuration file path
  nPrintResolution    : LREAL;                // printhead print resolution
  nSubPixelResolution : LREAL;                // position subpx resolution
  sPHType             : ST_PH_DEF; 						// Printhead hw type definition
  ePcType             : E_PcTypes;            // PrintController hw type
  nPcYShiftCenterRam  : UDINT;                // PrintController Y-Shift for centering in RAM (memory section configuration)
  fPhTempDeviation    : LREAL := 1.0;         // ph temperature deviation [°C] from setpoint to generate error (abs), default= +/- 1°C
END_STRUCT
END_TYPE

// ---- POUs/Print/Module/ST_MappingDefinition.TcDUT
(*
  Hardware mapping definition.
*)
TYPE ST_MappingDefinition :
STRUCT
  // absolute hw mapping
  nPhInst : UDINT := 1;      // ph hw instance selection
  nPcInst : UDINT := 1;      // pc hw instance selection
  nPgAbs  : UDINT := 1;      // absolute pg (eq PrintLine)
  // module internal mapping (relative to given nPm)
  nPm     : UDINT := 1;      // to pm x
  nPg     : UDINT := 1;      // to pg in pm x
  nPa     : UDINT := 1;      // to pa in pg
  nPs     : UDINT := 1;      // to ps in pa
  nPc     : UDINT := 1;      // to pc in pm
  nPcCh   : UDINT := 1;      // to pc channel of pc 1-4
END_STRUCT
END_TYPE

// ---- POUs/Print/Module/ST_ModuleMachineInterface_IN.TcDUT
TYPE ST_ModuleMachineInterface_IN :
STRUCT
  // Inputs (from machine)
  bEStop                            : BOOL;             // EStop active
  bSleep                            : BOOL;             // Sleep active
  bShutdown                         : BOOL;             // Shutdown active
  bMachineCommErr                   : BOOL;             // Machine communication error
  bSafetyCoverOk                    : BOOL;             // Safety cover OK (closed)
  bServiceDoorsOk                   : BOOL;             // Safety Doors OK (closed)
  bSafetyOk                         : BOOL;             // generic safety hardware ok
  bDriftControlError                : BOOL;             // (obsolete) remove?
  bDriftControlMissMarks            : BOOL;             // (obsolete) remove?
  
  // new
  bUnitInPrintPosition              : BOOL;             // Print module in print position
  bUnitInMaintPosition              : BOOL;             // Print module in maintenance position
  bUnitInCappingPosition            : BOOL;             // Print module in capping position
  bEngaged                          : BOOL;             // Print module engaged
  bPrintActivated                   : BOOL;             // Printing enabled (PrintON)
  bStopRequest                      : BOOL;             // Synced print stop, finish printing current actual repeat
  bFastStopRequest                  : BOOL;             // Fast print stop request
  bPrintDirection                   : BOOL;             // normal = 0, reverse = 1
  
  // other
  fSubstrateThickness               : LREAL := 0.000_1; // Substrate thickness [m]
  fSubstrateLen                     : LREAL;            // Substrate length [m]
  fSubstrateWidth                   : LREAL;            // Substrate width [m]
  fWebStretchCalculated             : LREAL;            // Web strech factor converted
  fLateralRegister                  : LREAL;            // Lateral regster [m]
  fDistanceToPrevModule             : LREAL;            // Distance to previous PrintModule [m] (dist to prev mark sensor, which is pm reference pos) 
  fInspectionDistToPrint            : LREAL;            // Inspection distance to PrintModule [m}
  bTargetSpeedReached               : BOOL;             // Target speed reached
  fTargetSpeed                      : LREAL;            // Target speed [m/s]
  bPrintMarkExist                   : BOOL;             // Print markus exist
  fMarkToPrintdataCenterY           : LREAL;            // mark distance from print data center Y [m]
  fMarkBaseSize                     : LREAL;            // mark base "a" size (square side) [m]
  fMarkDistToStartMark              : LREAL;            // mark distance repeat to start mark [m}
  nUsePerRepeatInLine               : UDINT;            // Number of Uses per Repead in printing direction
  
  fEncoderResolution                : LREAL;            // Effective Encoder resolution to be used [pulse/um]
  fEncoderDetectPulseMin            : LREAL;            // Encoder step measurement minimum pulse 
  fEncoderDetectPulseMax            : LREAL;            // Encoder step measurement maximum pulse
  nEncoderDetectFilterSz            : UDINT;            // Mean filter size for measured encoder pulse output
  
  nDistanceSheetDetIMCToNip_um      : UDINT;            // Distance from SheetDetection IMC to Nip [µm]
  nDistanceSheetDetCRToNip_um       : UDINT;            // Distance from SheetDetection CodeReader to Nip [µm]
  nDistanceSheetDetCoronaToNip_um   : UDINT;            // Distance from SheetDetection Corona to Nip [µm]
  nDistanceSheetDetPrintToNip_um    : UDINT;            // Distance from SheetDetection StartEdgePrintLine to Nip [µm]
  bMaintenanceActive                : BOOL;             // Z-Axis is on Position Maintenance and the Ink-Jet Tub is in Service Position
  nMachineType                      : UDINT;            // 0 = DM-Maxliner 3D B1 (dmax), 1 = DM-Uniliner (Concept 4), 2, 3 = DM-Maxliner 2D B3, DM-Maxliner 2D B2 (BigBob)
END_STRUCT
END_TYPE

// ---- POUs/Print/Module/ST_ModuleMachineInterface_OUT.TcDUT
TYPE ST_ModuleMachineInterface_OUT :
STRUCT
  // Outputs (to Machine)
  // -- from Print
  bMoving               : BOOL;             // substrate/module is moving
  fSpeed                : LREAL;            // Current module speed [m/s]
  fPosition             : LREAL;            // PrintPostion [m]
  fMaxSpeed             : LREAL;            // Max. possible print module speed [m/s]
  bLengthMismatch       : BOOL;             // image/format length mismatch
  bStopReady            : BOOL;             // Module is ready to stop moving (for synced stop)
  bSpeedExeeded         : BOOL;             // Module speed exeeded
  fHeadGap              : LREAL;            // Head gap from PUC [m] (from Ads SA converted)
  fInkQuantity          : LREAL;            // InkQuantity (from Ads PG)
  fEncoderStepsMeasured : LREAL;            // Measured encoder pulse between the effective encoder step measurement [pulse]
END_STRUCT
END_TYPE

// ---- POUs/Print/obsolete/ST_CassetteSetup_PrintAds.TcDUT
TYPE ST_CassetteSetup_PrintAds :
STRUCT

  aPM_Name : STRING[10];
  aPG_Name : ARRAY[1..GVL_WEU.nC_MaxWorkerPrintPerPm] OF STRING[22];
  aPC_Name : ARRAY[1..GVL_WEU.nC_MaxPcPerPm] OF STRING[22];
  aPH_Name : ARRAY[1..GVL_WEU.nC_MaxPhPerPm] OF STRING[15];
  
{IF defined (Production_1PM)}

  aC_PM_NAME                    : ARRAY[1..iCPr_NB_PM] OF STRING[10] :=
           ['Module 3'];

  aC_PG_NAME                    : ARRAY[1..iCPr_NB_PM] OF ARRAY[1..iCPr_NB_PG] OF STRING[22] := [
            ['M3 Printline 1 infeed', 'M3 Printline 2 outlet']];  // PM1

  aC_PC_NAME                    : ARRAY[1..iCPr_NB_PC] OF STRING[22] :=
           ['Controller Board 1.1',
            'Controller Board 1.2',
            'Controller Board 2.1',
            'Controller Board 2.2'];

  aC_PH_NAME                    : ARRAY[1..iCPr_NB_PH] OF STRING[15] :=
           ['Printhead 1.1',
            'Printhead 1.2',
            'Printhead 1.3',
            'Printhead 1.4',
            'Printhead 1.5',
            'Printhead 1.6',
            'Printhead 2.1',
            'Printhead 2.2',
            'Printhead 2.3',
            'Printhead 2.4',
            'Printhead 2.5',
            'Printhead 2.6'];

{ELSE}

  aC_PM_NAME                    : ARRAY[1..iCPr_NB_PM] OF STRING[10] :=
           ['Module 3',
            'Module 4'];

  aC_PG_NAME                    : ARRAY[1..iCPr_NB_PM] OF ARRAY[1..GVL_WEU.nC_MaxWorkerPrintPerPm] OF STRING[22] := [
            ['M3 Printline 1 infeed', 'M3 Printline 2 outlet'],   // PM1
            ['M4 Printline 3 infeed', 'M4 Printline 4 outlet']];  // PM2

  aC_PC_NAME                    : ARRAY[1..iCPr_NB_PC] OF STRING[22] :=
           ['Controller Board 1.1',
            'Controller Board 1.2',
            'Controller Board 2.1',
            'Controller Board 2.2',
            'Controller Board 3.1',
            'Controller Board 3.2',
            'Controller Board 4.1',
            'Controller Board 4.2'];

  aC_PH_NAME                    : ARRAY[1..iCPr_NB_PH] OF STRING[15] :=
           ['Printhead 1.1',
            'Printhead 1.2',
            'Printhead 1.3',
            'Printhead 1.4',
            'Printhead 1.5',
            'Printhead 1.6',
            'Printhead 2.1',
            'Printhead 2.2',
            'Printhead 2.3',
            'Printhead 2.4',
            'Printhead 2.5',
            'Printhead 2.6',
            'Printhead 3.1',
            'Printhead 3.2',
            'Printhead 3.3',
            'Printhead 3.4',
            'Printhead 3.5',
            'Printhead 3.6',
            'Printhead 4.1',
            'Printhead 4.2',
            'Printhead 4.3',
            'Printhead 4.4',
            'Printhead 4.5',
            'Printhead 4.6'];

{END_IF}
 
  (*ADS configurations*)
  // PM 
  aC_GENERALSHIFT_X_UNIT          : STRING  :=
  lL_GENERALSHIFT_X_SET_MIN       : DINT    :=   -380_000;     (*minimum set value*)
  lL_GENERALSHIFT_X_SET_MAX       : DINT    :=  1_000_000;     (*maximum set value*)
  aC_GENERALSHIFT_Y_UNIT          : STRING  := 'um';
  lL_GENERALSHIFT_Y_SET_MIN       : DINT    := -8_001;         (*minimum set value*)
  lL_GENERALSHIFT_Y_SET_MAX       : DINT    :=  8_001;         (*maximum set value*)
  
  // PG
  aC_xx_STARTPOS_X_TYPE           : STRING  := 'DINT';
  aC_xx_STARTPOS_X_UNIT           : STRING  := 'um';
  lL_xx_STARTPOS_X_SET_MIN        : DINT    := 0;              (*minimum set value*)
  lL_xx_STARTPOS_X_SET_MAX        : DINT    := 2_000_000;      (*maximum set value*)
  aC_xx_STARTPOS_Y_UNIT           : STRING  := 'pixel';
  lL_xx_STARTPOS_Y_SET_MIN        : DINT    := 0;              (*minimum set value*)
  lL_xx_STARTPOS_Y_SET_MAX        : DINT    := 2147483647;     (*maximum set value*)
  
END_STRUCT
END_TYPE

// ---- GVLs/EC_DefGrid.TcGVL
{attribute 'qualified_only'}
(*
  Calmar Error Codes - CalmarProductsSteinemann library
*)
VAR_GLOBAL
  // base
  _ecBase        : UDINT := CalmarCommons.ErrorCodes.lCalmar_base;
  _ecProjBase    : UDINT := _ecBase OR 16#00150000;

  // DefGrid error
  ecDefGrid_DefGridError : T_ErrDef(Id:=_ecProjBase OR 16#001, Code:='GridError', Desc:='Error in script happened');
  ecDefGrid_DefGridAbort : T_ErrDef(Id:=_ecProjBase OR 16#002, Code:='GridAbort', Desc:='Deformation aborted');
  
  // Camera errors
  ecDefGrid_CamNotAvailable : T_ErrDef(Id:=_ecProjBase OR 16#010, Code:='CamNotAvailable', Desc:='Desired camera not available');
  
  // end (verify to not overflow the group range!)
END_VAR

// ---- GVLs/GVL_Camera.TcGVL
{attribute 'qualified_only'}
VAR_GLOBAL CONSTANT
  cMaxNbMarks                   : UDINT := 200;     (*Max number of QualiVision marks*)
  cMaxNbSectors                 : UDINT := 50;      (*Max number of QualiVision sectors*)
  cC_QUALIVISION_MAX_NB_MARKS   : BYTE  := 10;      (*Max number of QualiVision marks*)
  nC_NbCamErrors                : UDINT := 10;
END_VAR

// ---- GVLs/GVL_Deformation.TcGVL
{attribute 'qualified_only'}
VAR_GLOBAL
// moved to CompPrint FB_PH
  //  nC_GridPitch_X  : UDINT := 1024;    // GRID: distance between grid point in y [px] (FPGA definition)
  //  nC_GridPitch_Y  : UDINT := 2048;    // GRID: distance between grid point in y [px] (FPGA definition)
  //  nC_GridRoiRows  : UINT  := 3;       // ROI: [1024=4,  2048=3] number of roi rows per head (FPGA definition) 
  //  nC_GridRoiCols  : UINT  := 85;      // ROI: [1024=62, 2048=85] number of roi columns per head (FPGA definition) 

  nC_DefaultGridPitch_X  : UDINT := 1024;    // GRID: (default if unknown in hw) distance between grid point in y [px] (FPGA definition)
  nC_DefaultGridPitch_Y  : UDINT := 2048;    // GRID: (default if unknown in hw) distance between grid point in y [px] (FPGA definition)
  nC_GridSubReso  : UDINT := 10;      // sub resolution of grid definitions (script handling)
  bC_UsePUDeformation : BOOL := TRUE;   // enable calculation of PU deformation/correction
END_VAR

// ---- GVLs/GVL_WEU.TcGVL
{attribute 'qualified_only'}
VAR_GLOBAL CONSTANT
  nC_MaxWorkerPrintPerPm  : UDINT := 2;
  nC_MaxPcPerPm           : UDINT := 10;
  nC_MaxPhPerPm           : UDINT := 40;
  
  fC_MaxMachineSpeed      : LREAL := TO_LREAL(100)/60;   // max module speed (100 m/min) in [m/s]
  
  // compensations
  nC_CurrentTimeStampComp : UDINT := 2_000;   // [us] current timestamp compensation for timestamp input
  nC_SensorTimeStampComp  : UDINT := 150;     // [us] time compensation for input edge
END_VAR

// ---- GVLs/GVL_Maxliner.TcGVL
{attribute 'qualified_only'}
VAR_GLOBAL CONSTANT
  nC_MaxWorkerPrintPerPm  : UDINT := 1;
  nC_MaxPcPerPm           : UDINT := 4;
  nC_MaxPhPerPm           : UDINT := 11;
  
  fC_MaxMachineSpeed      : LREAL := TO_LREAL(100)/60;   // max module speed (100 m/min) in [m/s]
  
  aC_PlcProjectCfgPath    : T_MaxString := 'C:\ProgramData\WifagPolytype\DMAXPrintUnitPlc\02_Plc\DP-ST-1044-Steinemann\Steinemann\PlcProject\Configuration\';

  // compensations
  nC_CurrentTimeStampComp : UDINT := 2_000;   // [us] current timestamp compensation for timestamp input
  nC_SensorTimeStampComp  : UDINT := 150;     // [us] time compensation for input edge
END_VAR

// ---- Version/Global_Version.TcGVL
{attribute 'TcGenerated'}
{attribute 'no-analysis'}
{attribute 'linkalways'}
// This function has been automatically generated from the project information.
VAR_GLOBAL CONSTANT
	{attribute 'const_non_replaced'}
	stLibVersion_CalmarProductSteinemann : ST_LibVersion := (iMajor := 3, iMinor := 0, iBuild := 4, iRevision := 0, nFlags := 0, sVersion := '3.0.4');
END_VAR

// ---- POUs/Machine/CleaningStation/I_CleanDevice.TcIO
INTERFACE I_CleanDevice

METHOD mAbort : BOOL
VAR_INPUT
END_VAR
END_METHOD

METHOD mAckError
VAR_INPUT
END_VAR
END_METHOD

METHOD mOperation : BOOL
VAR_INPUT
	iI_Step : INT;
END_VAR
END_METHOD

METHOD mSetMode : BOOL
VAR_INPUT
	sI_CleanMode : EN_CLEANING_OP;
END_VAR
END_METHOD

PROPERTY sStatus : ST_CLEANING_DEV_STATUS
GET
END_GET
END_PROPERTY

END_INTERFACE

// ---- POUs/Machine/CleaningStation/I_CleaningStateCallback.TcIO
INTERFACE I_CleaningStateCallback

METHOD mChangeState
VAR_INPUT
	sI_NextState : EN_Cleaning_State;
END_VAR
END_METHOD

METHOD mDeviceAbort : BOOL
VAR_INPUT
END_VAR
END_METHOD

METHOD mDeviceAckError
VAR_INPUT
END_VAR
END_METHOD

METHOD mDeviceOperation : BOOL
VAR_INPUT
	iI_Step : INT;	
END_VAR
END_METHOD

METHOD mSetMode : BOOL
VAR_INPUT
	sI_CleanMode	: EN_CLEANING_OP;
END_VAR
END_METHOD

PROPERTY pDeviceStatus : ST_CLEANING_DEV_STATUS
GET
END_GET
END_PROPERTY

END_INTERFACE

// ---- POUs/Machine/CleaningStation/I_MachineState.TcIO
INTERFACE I_MachineState EXTENDS I_MachineStateBase

PROPERTY pError : BOOL
GET
END_GET
END_PROPERTY

PROPERTY pMaintenance : BOOL
GET
END_GET
END_PROPERTY

PROPERTY pProduction : BOOL
GET
END_GET
END_PROPERTY

PROPERTY pSleep : BOOL
GET
END_GET
END_PROPERTY

END_INTERFACE

// ---- POUs/Machine/CleaningStation/I_MachineStateBase.TcIO
INTERFACE I_MachineStateBase

PROPERTY pMachineReady : BOOL
GET
END_GET
END_PROPERTY

PROPERTY pSafetyOk : BOOL
GET
END_GET
END_PROPERTY

END_INTERFACE

// ---- POUs/Print/Camera/I_Camera.TcIO
INTERFACE I_Camera

METHOD ActivateCam : BOOL
VAR_INPUT
  iCameraSink : I_CameraSink;
END_VAR
END_METHOD

(*
  Activate/Deactivate camera trigger device
*)
PROPERTY bEnableTrigger : BOOL
SET
END_SET
END_PROPERTY

(*
  Activate/Deactivate camera manual teach mode
*)
PROPERTY bManualTeach : BOOL
SET
END_SET
END_PROPERTY

{attribute 'monitoring':='call'}
PROPERTY bSimulate : BOOL
GET
END_GET
SET
END_SET
END_PROPERTY

METHOD DeactivateCam : BOOL
VAR_INPUT
  iSink : I_CameraSink;
END_VAR
END_METHOD

{attribute 'monitoring':='call'}
PROPERTY ABSTRACT eCameraMode : E_CameraMode
GET
END_GET
END_PROPERTY

{attribute 'monitoring':='call'}
PROPERTY ABSTRACT eDeviceType : E_CameraDevice
GET
END_GET
END_PROPERTY

{attribute 'monitoring':='call'}
PROPERTY fCameraToPrintOffset : LREAL
GET
END_GET
END_PROPERTY

{attribute 'monitoring':='call'}
PROPERTY fDetectToCameraOffset : LREAL
GET
END_GET
END_PROPERTY

{attribute 'monitoring':='call'}
// camera frame size in [px]
PROPERTY fFrameLength : LREAL
GET
END_GET
SET
END_SET
END_PROPERTY

{attribute 'monitoring':='call'}
(*Image Length/Depth in [m]*)
PROPERTY fImageLength : LREAL
GET
END_GET
SET
END_SET
END_PROPERTY

{attribute 'monitoring':='call'}
(*Image Width in [m]*)
PROPERTY fImageWidth : LREAL
GET
END_GET
SET
END_SET
END_PROPERTY

{attribute 'monitoring':='call'}
(*Substrate Length/Depth in [m]*)
PROPERTY fSubstrateLength : LREAL
GET
END_GET
SET
END_SET
END_PROPERTY

{attribute 'monitoring':='call'}
(*Substrate Width in [m]*)
PROPERTY fSubstrateWidth : LREAL
GET
END_GET
SET
END_SET
END_PROPERTY

{attribute 'monitoring':='call'}
PROPERTY fTriggerDistance : LREAL
GET
END_GET
SET
END_SET
END_PROPERTY

(*
  Get camera status.
  :return: TRUE if camera is ok
*)
METHOD GetCamStatus : BOOL  // Camera Ok?
VAR_OUTPUT
  bConnectionOK  : BOOL;    // Camera connected
  bTeachOk       : BOOL;    // Teach successful
  nTeachedPoints : UDINT;   // Teached points for this job
  nScannedPoints : UDINT;   // Scanned points on current CT
  bCamStarted    : BOOL;    // Camera trigger is active, cam started
  bCamDone       : BOOL;    // Camera finished on last CT
  bErrors        : ARRAY[1..GVL_Camera.nC_NbCamErrors] OF BOOL;  // generic error flag list
END_VAR
END_METHOD

METHOD mJobStart : BOOL
VAR_INPUT
END_VAR
END_METHOD

(*
  Set mode to camera.
  :return: TRUE if success
*)
METHOD setCameraMode : BOOL
VAR_INPUT
  eCameraMode : E_CameraMode;
END_VAR
END_METHOD

METHOD setMsgInterface : BOOL
VAR_INPUT
  pMsgConfig  : POINTER TO ST_MSG_CONFIG;
END_VAR
END_METHOD

{attribute 'monitoring':='call'}
PROPERTY sName : STRING
GET
END_GET
END_PROPERTY

{attribute 'monitoring':='call'}
PROPERTY sVisuName : STRING
GET
END_GET
END_PROPERTY

END_INTERFACE

// ---- POUs/Print/Camera/I_CameraSink.TcIO
{attribute 'monitoring':='call'}
INTERFACE I_CameraSink

METHOD AddCamPoint : BOOL
VAR_INPUT
	sDeformationPoint	: ST_DeformationPointAccurate;
END_VAR
END_METHOD

METHOD AddTeachPoint : BOOL
VAR_INPUT
  sTeachPoint : ST_DeformationPointAccurate;
END_VAR
END_METHOD

(*
  Event cam done "detecting points", sheet/repeate done.
  Called after last point will be streamed to same CT.
*)
METHOD CamDone : BOOL
END_METHOD

(*
  Event cam started "detecting points".
  Is called before streaming cam points.
*)
METHOD CamStarted
VAR_INPUT
  nX0 : DINT; // detected start position
END_VAR
END_METHOD

// Detected "real" image lenght [m]
PROPERTY fPrintLengthEffective : LREAL
SET
END_SET
END_PROPERTY

END_INTERFACE

// ---- POUs/Print/Camera/I_CameraTrigger.TcIO
INTERFACE I_CameraTrigger

PROPERTY bManualTeach : BOOL
GET
END_GET
SET
END_SET
END_PROPERTY

METHOD Disable : BOOL
VAR_INPUT
END_VAR
END_METHOD

METHOD Enable : BOOL
VAR_INPUT
  iCam : I_CameraTriggerDevice;
  bUseCameraTrigger : BOOL; //Generate camera trigger
  bUseCameraTriggerFeedback : BOOL; //Use feedback as trigger?
END_VAR
END_METHOD

METHOD SetSubstrateLength
VAR_INPUT
  fSubstrateLength : LREAL;
END_VAR
END_METHOD

END_INTERFACE

// ---- POUs/Print/Camera/I_CameraTriggerDevice.TcIO
INTERFACE I_CameraTriggerDevice

METHOD CamTrigger
VAR_INPUT
  bOk             : BOOL;     // trigger is ok
	nPos            : DINT;     // camera triggered position
  nPosDeviation   : DINT;     // camera started deviation
  nX0             : DINT;     // detected position sheet/repetition
END_VAR
END_METHOD

METHOD CamTriggerDone
VAR_INPUT
END_VAR
END_METHOD

{attribute 'monitoring':='call'}
PROPERTY fTriggerDistance : LREAL
GET
END_GET
END_PROPERTY

PROPERTY fTriggerPulseLength : LREAL
GET
END_GET
END_PROPERTY

END_INTERFACE

// ---- POUs/Print/DefGrid/I_DeformationHandler.TcIO
INTERFACE I_DeformationHandler

METHOD DeleteCachedCt : BOOL
VAR_INPUT
  iCT              : I_CT;
END_VAR
END_METHOD

END_INTERFACE

// ---- POUs/Print/DefGrid/I_GridPointCorrection.TcIO
INTERFACE I_GridPointCorrection

(*
  Apply correction to gridPoint
*)
METHOD updateCorrection : BOOL
VAR_INPUT
  pPoint : POINTER TO ST_DeformationPointAccurate;
END_VAR
END_METHOD

END_INTERFACE

// ---- POUs/Print/DefGrid/I_Module.TcIO
INTERFACE I_Module

{attribute 'monitoring' := 'call'}
PROPERTY bEstop : BOOL
GET
END_GET
SET
END_SET
END_PROPERTY

{attribute 'monitoring' := 'call'}
PROPERTY bSleep : BOOL
GET
END_GET
SET
END_SET
END_PROPERTY

(*
  Register to get Emergency state updates.
*)
METHOD registerForEmergencyUpdate : BOOL
VAR_INPUT
	iObserver	: I_EmergencyObserver;
END_VAR
END_METHOD

(*
  Register to get sleep state updates.
*)
METHOD registerForSleepUpdate : BOOL
VAR_INPUT
	iObserver	: I_SleepObserver;
END_VAR
END_METHOD

END_INTERFACE

// ---- POUs/Print/DefGrid/I_ParamMediator.TcIO
INTERFACE I_ParamMediator

PROPERTY sCameraGridSettings : ST_CameraGridSettings
GET
END_GET
END_PROPERTY

PROPERTY sDeformationGridSettings : ST_DefGridSettings
GET
END_GET
END_PROPERTY

END_INTERFACE

// ---- POUs/Print/DefGrid/I_ProdManager.TcIO
INTERFACE I_ProdManager

END_INTERFACE

// ---- POUs/Print/Global/I_PrintGlobal.TcIO
INTERFACE I_PrintGlobal

PROPERTY iHardwarePool : I_HardwarePool
GET
END_GET
END_PROPERTY

PROPERTY iMasterPrintPosition : I_PrintPosition
GET
END_GET
END_PROPERTY

(*
  Register for PU StatusClient
*)
METHOD registerPuStatusClient : BOOL
VAR_INPUT
  sClient       : I_PrintStatusClient;
END_VAR
END_METHOD

METHOD registerPuSubystem : BOOL
VAR_INPUT
  iSubSys      : I_PrintSubsystem;
END_VAR
END_METHOD

END_INTERFACE

// ---- POUs/Machine/CleaningStation/ADS/FB_ADS_CleanAxis.TcPOU
FUNCTION_BLOCK FB_ADS_CleanAxis EXTENDS FB_AdsBlockBase
VAR
  // ---------------------------------
  // ADS interface block specific
  sO_Message            : ST_ADS_MSG_IF;    (*Messaging*)

  bI_FaultAck           : BOOL := FALSE;

  (*Manual Move, only possible when in maintenance and manual mode*)
  bI_ManualMove         : BOOL := FALSE;  (*Active as long as true*)
  bO_ManualMoveCanEx    : BOOL := FALSE;
  bO_ManualMovekExec    : BOOL := FALSE;
  fI_ManualTargetPos    : REAL := 0.0;

  (*Current axis position*)
  sO_AxisPosition       : ST_VAR_OUT_REAL;

  wO_ErrorCode          : WORD;
  bO_Busy               : BOOL;
  bO_Ready              : BOOL;
  bO_Error              : BOOL;
END_VAR

VAR PERSISTENT
  nR_Pattern            : UDINT;  (*check pattern for rem validity*)
END_VAR

METHOD config
VAR_INPUT
  aName               : STRING;
  sAxisPositionUnit   : STRING;  
  fAxisPositionMin    : REAL;  
  fAxisPositionMax    : REAL;  
END_VAR
aO_Name                  := aName;

sO_AxisPosition.bC_Exist := TRUE; 
sO_AxisPosition.aC_Unit  := sAxisPositionUnit; 
sO_AxisPosition.fC_Min   := fAxisPositionMin; 
sO_AxisPosition.fC_Max   := fAxisPositionMax; 

(*OPC-UA: EngineeringUnits*)
sO_AxisPosition.nC_EngineeringUnits := 5066068;  (*[mm]*)
END_METHOD

METHOD PROTECTED initRemVar
VAR_INPUT
END_VAR
(*load default initial values if pattern was invalid*)
IF nR_Pattern <> 16#ABCD THEN
  ;
ELSE  
  nR_Pattern      := 16#ABCD;
END_IF

(*Init values*)
END_METHOD

METHOD ResetCommands : BOOL
VAR_INPUT
END_VAR
bI_ManualMove := FALSE;
END_METHOD

METHOD setFeedback
VAR_INPUT
  bManualMoveCanEx         : BOOL; 
  bManualMovekExec         : BOOL;  

  fAxisPositionVal         : REAL;  

  wErrorCode               : WORD; 
  bBusy                    : BOOL; 
  bReady                   : BOOL; 
  bError                   : BOOL; 
END_VAR
bO_ManualMoveCanEx         := bManualMoveCanEx;
bO_ManualMovekExec         := bManualMovekExec;

sO_AxisPosition.fO_Val     := fAxisPositionVal;

wO_ErrorCode               := wErrorCode;
bO_Busy                    := bBusy;
bO_Ready                   := bReady;
bO_Error                   := bError;
END_METHOD

(*
  Setup constant ADS Block definitions.
  HOWTO: in abstract implmentation call
      init(aVersion:=, aType:=, nType:=, eLayer:=);
*)
METHOD  setup
init( aVersion := '01.00.01'
    , aType    := 'CleanAxis'
    , nType    := eMa_BLK_MACHINE
    , eLayer   := E_AdsLayer.Structural);
END_METHOD

PROPERTY sMsgInterface : POINTER TO ST_ADS_MSG_IF
GET
sMsgInterface := ADR(sO_Message);
END_GET
END_PROPERTY

END_FUNCTION_BLOCK

// ---- POUs/Machine/CleaningStation/ADS/FB_ADS_CleanProcess.TcPOU
FUNCTION_BLOCK FB_ADS_CleanProcess EXTENDS FB_AdsBlockBase
VAR
  // ---------------------------------
  // ADS interface block specific
  sO_Message                 : ST_ADS_MSG_IF;    (*Messaging*)

  (*User commands - Trigger operation*)
  bI_StartCapping            : BOOL := FALSE;
  bO_StartCappingCanEx       : BOOL := FALSE;
  bO_StartCappingExec        : BOOL := FALSE;
                             
  bI_StopCapping             : BOOL := FALSE;
  bO_StopCappingCanEx        : BOOL := FALSE;
  bO_StopCappingExec         : BOOL := FALSE;
                             
  bI_Purge                   : BOOL := FALSE;
  bO_PurgeCanEx              : BOOL := FALSE;
  bO_PurgeExec               : BOOL := FALSE;
                             
  bI_Clean                   : BOOL := FALSE;
  bO_CleanCanEx              : BOOL := FALSE;
  bO_CleanExec               : BOOL := FALSE;
                             
  bI_Maintenance             : BOOL := FALSE;
  bO_MaintenanceCanEx        : BOOL := FALSE;
  bO_MaintenanceExec         : BOOL := FALSE;
                             
  bI_OpenShutter             : BOOL := FALSE;
  bO_OpenShutterCanEx        : BOOL := FALSE;
  bO_OpenShutterExec         : BOOL := FALSE;
                             
  bI_Abort                   : BOOL := FALSE;
  bO_AbortCanEx              : BOOL := FALSE;
  bO_AbortExec               : BOOL := FALSE;

  bI_AcknowledgeError        : BOOL := FALSE;
  bO_AcknowledgeErrorCanEx   : BOOL := FALSE;
  bO_AcknowledgeErrorExec    : BOOL := FALSE;

  (*User settings - State operation*)
  bI_AutoMode                : BOOL := TRUE;  (*del*)
  bI_CleanAfterCapp          : BOOL := FALSE;
  bI_CleanAfterPurge         : BOOL := FALSE;
  bI_PurgeAfterCapp          : BOOL := FALSE; (*del*)
  bI_MaintenanceMode         : BOOL := FALSE;
                             
  (*Flags*)                  
  bO_Busy                    : BOOL;
  bO_Ready                   : BOOL;
  bO_ServiceEnabled          : BOOL;
  bO_AxisProcessMovingVisible: BOOL := TRUE;  (*Cleaning process axis moving is shown at PUC*)
                             
  (*Message Queue - TODO update*)
  bI_FaultAck                : BOOL := FALSE;
  wO_ErrorCode               : WORD;
END_VAR

VAR PERSISTENT
  nR_Pattern                 : UDINT;  (*check pattern for rem validity*)
END_VAR

PROPERTY bAcknowledgeError : BOOL
SET
bI_AcknowledgeError := bAcknowledgeError;
END_SET
END_PROPERTY

METHOD config
VAR_INPUT
  aName                     : STRING;
  bAxisProcessMovingVisible : BOOL;  
END_VAR
aO_Name                     := aName;

bO_AxisProcessMovingVisible := bAxisProcessMovingVisible;
END_METHOD

METHOD PROTECTED initRemVar
VAR_INPUT
END_VAR
(*load default initial values if pattern was invalid*)
IF nR_Pattern <> 16#ABCD THEN
  ;
ELSE  
  nR_Pattern      := 16#ABCD;
END_IF

(*Init values*)
END_METHOD

METHOD ResetCommands : BOOL
VAR_INPUT
END_VAR
bI_StartCapping := FALSE;
bI_StopCapping  := FALSE;
bI_Maintenance  := FALSE;
bI_Clean        := FALSE;
bI_Purge        := FALSE;
END_METHOD

METHOD setFeedback
VAR_INPUT
  bStartCappingCanEx       : BOOL; 
  bStartCappingExec        : BOOL;  

  bStopCappingCanEx        : BOOL;  
  bStopCappingExec         : BOOL;  

  bPurgeCanEx              : BOOL; 
  bPurgeExec               : BOOL;  

  bCleanCanEx              : BOOL; 
  bCleanExec               : BOOL;  

  bMaintenanceCanEx        : BOOL;  
  bMaintenanceExec         : BOOL;  

  bOpenShutterCanEx        : BOOL;  
  bOpenShutterExec         : BOOL;  

  bAbortCanEx              : BOOL; 
  bAbortExec               : BOOL;  

  bAcknowledgeErrorCanEx   : BOOL;  
  bAcknowledgeErrorExec    : BOOL;  

  bBusy                    : BOOL; 
  bReady                   : BOOL; 
  bServiceEnabled          : BOOL; 
  bAxisProcessMovingVisible: BOOL; 

  wErrorCode               : WORD; 
END_VAR
bO_StartCappingCanEx       := bStartCappingCanEx;
bO_StartCappingExec        := bStartCappingExec;

bO_StopCappingCanEx        := bStopCappingCanEx;
bO_StopCappingExec         := bStopCappingExec;

bO_PurgeCanEx              := bPurgeCanEx;
bO_PurgeExec               := bPurgeExec;

bO_CleanCanEx              := bCleanCanEx;
bO_CleanExec               := bCleanExec;

bO_MaintenanceCanEx        := bMaintenanceCanEx;
bO_MaintenanceExec         := bMaintenanceExec;

bO_OpenShutterCanEx        := bOpenShutterCanEx;
bO_OpenShutterExec         := bOpenShutterExec;

bO_AbortCanEx              := bAbortCanEx;
bO_AbortExec               := bAbortExec;

bO_AcknowledgeErrorCanEx   := bAcknowledgeErrorCanEx;
bO_AcknowledgeErrorExec    := bAcknowledgeErrorExec;

bO_Busy                    := bBusy;
bO_Ready                   := bReady;
bO_ServiceEnabled          := bServiceEnabled;
bO_AxisProcessMovingVisible:= bAxisProcessMovingVisible;

wO_ErrorCode               := wErrorCode;
END_METHOD

(*
  Setup constant ADS Block definitions.
  HOWTO: in abstract implmentation call
      init(aVersion:=, aType:=, nType:=, eLayer:=);
*)
METHOD  setup
init( aVersion := '01.00.01'
    , aType    := 'CleanProcess'
    , nType    := eMa_BLK_MACHINE
    , eLayer   := E_AdsLayer.Structural);
END_METHOD

PROPERTY sMsgInterface : POINTER TO ST_ADS_MSG_IF
GET
sMsgInterface := ADR(sO_Message);
END_GET
END_PROPERTY

END_FUNCTION_BLOCK

// ---- POUs/Machine/CleaningStation/FB_CappingCommand.TcPOU
FUNCTION_BLOCK FB_CappingCommand

VAR_INPUT
  IbTrigger                                 : BOOL;
  IbReset                                   : BOOL;
END_VAR

VAR_OUTPUT
  ObCappingCommand                          : BOOL;
END_VAR

VAR
  fb_TonTrigger                             : TON;
  fb_TonReset                               : TON;
  bL_CappingCommandAfterEngaged             : BOOL;
END_VAR

VAR CONSTANT
  tC_DELAY_CAPPING_COMMAND                  : TIME := T#500MS;    (*Delay for automatic generated capping commands*)
  tC_RELEASE_CAPPING_COMMAND                : TIME := T#2S;       (*Release for automatic generated capping commands*)
END_VAR

fb_TonTrigger(IN := IbTrigger, PT := tC_DELAY_CAPPING_COMMAND);
IF fb_TonTrigger.Q THEN
  ObCappingCommand := TRUE;
END_IF
fb_TonReset(IN := IbTrigger, PT := tC_RELEASE_CAPPING_COMMAND);
IF fb_TonReset.Q OR IbReset THEN
  ObCappingCommand := FALSE;
END_IF

END_FUNCTION_BLOCK

// ---- POUs/Machine/CleaningStation/FB_CH_MOTION_CTRL.TcPOU
FUNCTION_BLOCK FB_CH_MOTION_CTRL
(******************************************************************************************)
(*  FILENAME:     FB_CH_MOTION_CTRL                                                       *)
(*  PROJECT:      Steinemann                                                              *)
(*  COPYRIGHT:    Wifag-Polytype                                                          *)
(*  ENVIRONMENT:  TwinCat2, v2.11                                                         *)
(*  VERSION:      1.0                                                                     *)
(*  DESCRIPTION:                                                                          *)
(*    This function pilots the mouvements of the Cleaning Head                            *)
(*    It checks the status of the Cleaning Unit and the Printer Unit                      *)
(*    to put the Cleaning Head in position and send command to it                         *)
(*  AUTHOR:      M: BOYRAZ, GoConcept                                                     *)
(******************************************************************************************)
(*	MODIFICATIONS:                                                                        *)
(******************************************************************************************)
(*  Date        Authtor   Descriptons                                                     *)
(*                                                                                        *)
(******************************************************************************************)

VAR_INPUT
  (*From Cleaning Head*)
  bI_ClnHeadEnabled          : BOOL;
  bI_ClnHeadError            : BOOL;

